// TwinCAT 3 PLC project JumpStart
// Title: Lift Template
// Company: FHNW
// Author: mbo
// ProjectVersion: 1.0.0
// ProgramVersion: 3.1.4026.20
// CompilerDefines: VISU_USEPROPERTYINFO
// libraries:
//   Tc2_Math, * (Beckhoff Automation GmbH)
//   Tc2_MC2, * (Beckhoff Automation GmbH)
//   Tc2_Standard, * (Beckhoff Automation GmbH)
//   Tc2_System, * (Beckhoff Automation GmbH)
//   Tc2_Utilities, * (Beckhoff Automation GmbH)
//   Tc3_IotBase, * (Beckhoff Automation GmbH)
//   Tc3_JsonXml, * (Beckhoff Automation GmbH)
//   VisuDialogs, * (System)
// project tree:
//   0_App/ IO_L1.TcGVL, IO_PLC.TcGVL, Divers.TcGVL, MAIN.TcPOU
//   0_App/Lib/Diverses/ ENUM_Achse.TcDUT, ENUM_Fahrsystem.TcDUT, ENUM_Tuer.TcDUT, FB_Logik_FIFO.TcPOU, FB_Logik_ShortestDistance.TcPOU, ITF_Fahrlogik.TcIO, ST_Error.TcDUT, ST_Fahrauftrag.TcDUT
//   0_App/Lib/ FB_Achse.TcPOU, FB_Blinker.TcPOU, FB_Fahrleitsystem.TcPOU, FB_Manuell.TcPOU, FB_Panel.TcPOU, FB_Taskmanager_1.TcPOU, FB_Tuer.TcPOU, FC_GetFloorPosition.TcPOU
//   7_Visu/Common/ Control.TcVIS, Floor.TcVIS, FloorControl.TcVIS, Lift.TcVIS, Lift_Axis.TcVIS, Lift_Floors.TcVIS, View_3Lifts.TcVIS
//   7_Visu/ Lift_1.TcVIS, Handbetrieb.TcVIS, Visu_Liftkabine.TcGVL, Visu_Liftkabine.TcVIS, Visu_Manuellmodus.TcGVL
//   9_Modell/Lib/ FB_MotionAxisPassive.TcPOU, FB_SimpleAxis.TcPOU, F_CycleTime.TcPOU, F_SpeedPerCycle.TcPOU
//   9_Modell/ MAIN_Modell.TcPOU, Visu_L1.TcGVL
//   / GlobalTextList.TcGTLO, PlcTask.TcTTO, Visualization Manager.TcVMO (not stored)
// real-time tasks:
//   TASK PlcTask: cycle T#10ms, priority 20, ADS port 350
// motion (NC):
//   TASK NC-Task 1 SAF: cycle T#2ms, priority 4, ADS port 501
//   TASK NC-Task 1 SVB: cycle T#10ms, priority 8, ADS port 511
//   AXIS Achse 1 - Lift1 (id 1)
//     Dynamic: Acceleration=1200, Deceleration=1200, Jerk=7200
//     Velo: FastManual=300, Maximum=500
//     OtherSettings: AllowMotionCmdToSlave=true
//     encoder EncType=4
//       EncPara: ScaleFactorNumerator=0.045066, MaxCount=#x0000ffff
//         Inc: RefSearchInverse=true, RefSyncInverse=false, RefMode=1, RefSoftSyncMask=#x0000ffff
//         TimeComp: TimeCompMode=1, EncDelayCycles=4
//     drive DrvType=23
//       DrvPara: Inverse=true
//         Analog: VeloReferenz=540, TorqueSetpointScale=10, ScaleFactorActTorque=0.1
//         TimeComp: TaskDelayCycles=1
//     controller CtrType=1
//       CtrPara: PriorControlFactor=1
//         PosDiffControl: Range=20
//         PID: PosKp=100
//         Observer: BandWidth=20
//   AXIS Achse 2 (id 2)
//     OtherSettings: AllowMotionCmdToSlave=true
//     encoder EncType=4
//       EncPara: MaxCount=#x0000ffff
//         Inc: RefSoftSyncMask=#x0000ffff
//     drive DrvType=23
//       Analog: TorqueSetpointScale=10, ScaleFactorActTorque=0.1
//       TimeComp: TaskDelayCycles=1
//     controller CtrType=1
//       CtrPara: PriorControlFactor=1
//         Observer: BandWidth=20
// I/O:
//   DEVICE Gerät 1 (EtherCAT), AmsNetId 192.168.10.51.2.1
//     Klemme 1 (EK1100) [EK1100 EtherCAT-Koppler (2A E-Bus)]
//       Klemme 2 (EL1262) [EL1262 2K. Dig. Eingang 24V, 1µs, DC Oversample]
//       Klemme 3 (EL2262) [EL2262 2K. Dig. Ausgang 24V, 1µs, DC Oversample]
//       Klemme 4 (EL1809) [EL1809 16K. Dig. Eingang 24V, 3ms]
//       Klemme 5 (EL2809) [EL2809 16K. Dig. Ausgang 24V, 0.5A]
//       Klemme 6 (EL3064) [EL3064 4K.Ana. Eingang 0-10V]
//       Klemme 7 (EL4004) [EL4004 4K. Ana. Ausgang 0-10V, 12bit]
//       Klemme 8 (EL5152) [EL5152 2K. Inc. Encoder]
//       Klemme 9 (EK1122) [EK1122 2-Port EtherCAT-Abzweig]
//       Klemme 10 (EL9011) [EL9011 Endklemme]
//   DEVICE Gerät 2 (EtherCAT), AmsNetId 192.168.10.51.3.1
//     Klemme 11 (EK1100) [EK1100 EtherCAT-Koppler (2A E-Bus)]
//       Klemme 12 (EL1809) [EL1809 16K. Dig. Eingang 24V, 3ms]
//       Klemme 13 (EL1809) [EL1809 16K. Dig. Eingang 24V, 3ms]
//       Klemme 14 (EL1809) [EL1809 16K. Dig. Eingang 24V, 3ms]
//       Klemme 15 (EL1809) [EL1809 16K. Dig. Eingang 24V, 3ms]
//       Klemme 16 (EL2809) [EL2809 16K. Dig. Ausgang 24V, 0.5A]
//       Klemme 17 (EL2809) [EL2809 16K. Dig. Ausgang 24V, 0.5A]
//       Klemme 18 (EL2809) [EL2809 16K. Dig. Ausgang 24V, 0.5A]
//       Klemme 19 (EL2809) [EL2809 16K. Dig. Ausgang 24V, 0.5A]
//       Klemme 20 (EL2809) [EL2809 16K. Dig. Ausgang 24V, 0.5A]
//       Klemme 21 (EL2809) [EL2809 16K. Dig. Ausgang 24V, 0.5A]
//       Klemme 22 (EL7342) [EL7342 2K. DC-Motor-Endstufe (50V, 3.5A)]
//       Klemme 37 (EL9011) [EL9011 Endklemme]
// variable links:
//   NC-Task 1 SAF/Axes/Achse 1 - Lift1 <-> Device 2 (EtherCAT)/Term 11 (EK1100)/Term 22 (EL7342)
//     Drive/Inputs/In/nState1 @bit 3 <-> DCM Status Channel 1/Status/Error
//     Drive/Inputs/In/nState1 @bit 5 <-> DCM Status Channel 1/Status/Moving negative
//     Drive/Inputs/In/nState1 @bit 4 <-> DCM Status Channel 1/Status/Moving positive
//     Drive/Inputs/In/nState1 @bit 1 <-> DCM Status Channel 1/Status/Ready
//     Drive/Inputs/In/nState1 <-> DCM Status Channel 1/Status/Ready to enable
//     Drive/Inputs/In/nState1 @bit 6 <-> DCM Status Channel 1/Status/Torque reduced
//     Drive/Inputs/In/nState1 @bit 2 <-> DCM Status Channel 1/Status/Warning
//     Drive/Inputs/In/nState2 @bit 4 <-> DCM Status Channel 1/Status/Digital input 2
//     Drive/Inputs/In/nState2 @bit 5 <-> DCM Status Channel 1/Status/Sync error
//     Drive/Inputs/In/nState2 @bit 7 <-> DCM Status Channel 1/Status/TxPDO Toggle
//     Drive/Inputs/In/nState4 @bit 1 <-> WcState/InputToggle
//     Drive/Inputs/In/nState4 <-> WcState/WcState
//     Drive/Outputs/Out/nCtrl1 <-> DCM Control Channel 1/Control/Enable
//     Drive/Outputs/Out/nCtrl1 @bit 2 <-> DCM Control Channel 1/Control/Reduce torque
//     Drive/Outputs/Out/nCtrl1 @bit 1 <-> DCM Control Channel 1/Control/Reset
//     Drive/Outputs/Out/nCtrl1 @bit 3 <-> DCM Control Channel 1/Control/Threshold active
//     Drive/Outputs/Out/nDataOut2[0] <-> DCM Velocity Channel 1/Velocity
//     Enc/Inputs/In/nDataIn1[0] <-> ENC Status compact Channel 1/Counter value
//     Enc/Inputs/In/nDataIn2[0] <-> ENC Status compact Channel 1/Latch value
//     Enc/Inputs/In/nState1 @bit 4 <-> ENC Status compact Channel 1/Status/Counter overflow
//     Enc/Inputs/In/nState1 @bit 3 <-> ENC Status compact Channel 1/Status/Counter underflow
//     Enc/Inputs/In/nState1 @bit 7 <-> ENC Status compact Channel 1/Status/Extrapolation stall
//     Enc/Inputs/In/nState1 @bit 1 <-> ENC Status compact Channel 1/Status/Latch extern valid
//     Enc/Inputs/In/nState1 @bit 2 <-> ENC Status compact Channel 1/Status/Set counter done
//     Enc/Inputs/In/nState2 @bit 4 <-> ENC Status compact Channel 1/Status/Status of extern latch
//     Enc/Inputs/In/nState2 <-> ENC Status compact Channel 1/Status/Status of input A
//     Enc/Inputs/In/nState2 @bit 1 <-> ENC Status compact Channel 1/Status/Status of input B
//     Enc/Inputs/In/nState2 @bit 5 <-> ENC Status compact Channel 1/Status/Sync error
//     Enc/Inputs/In/nState2 @bit 7 <-> ENC Status compact Channel 1/Status/TxPDO Toggle
//     Enc/Inputs/In/nState4 @bit 1 <-> WcState/InputToggle
//     Enc/Inputs/In/nState4 <-> WcState/WcState
//     Enc/Outputs/Out/nCtrl1 @bit 3 <-> ENC Control compact Channel 1/Control/Enable latch extern on negative edge
//     Enc/Outputs/Out/nCtrl1 @bit 1 <-> ENC Control compact Channel 1/Control/Enable latch extern on positive edge
//     Enc/Outputs/Out/nCtrl1 @bit 2 <-> ENC Control compact Channel 1/Control/Set counter
//     Enc/Outputs/Out/nDataOut1[0] <-> ENC Control compact Channel 1/Set counter value
//   NC-Task 1 SAF/Axes/Achse 2 <-> Device 2 (EtherCAT)/Term 11 (EK1100)/Term 22 (EL7342)
//     Drive/Inputs/In/nState1 @bit 3 <-> DCM Status Channel 2/Status/Error
//     Drive/Inputs/In/nState1 @bit 5 <-> DCM Status Channel 2/Status/Moving negative
//     Drive/Inputs/In/nState1 @bit 4 <-> DCM Status Channel 2/Status/Moving positive
//     Drive/Inputs/In/nState1 @bit 1 <-> DCM Status Channel 2/Status/Ready
//     Drive/Inputs/In/nState1 <-> DCM Status Channel 2/Status/Ready to enable
//     Drive/Inputs/In/nState1 @bit 6 <-> DCM Status Channel 2/Status/Torque reduced
//     Drive/Inputs/In/nState1 @bit 2 <-> DCM Status Channel 2/Status/Warning
//     Drive/Inputs/In/nState2 @bit 3 <-> DCM Status Channel 2/Status/Digital input 1
//     Drive/Inputs/In/nState2 @bit 4 <-> DCM Status Channel 2/Status/Digital input 2
//     Drive/Inputs/In/nState2 @bit 5 <-> DCM Status Channel 2/Status/Sync error
//     Drive/Inputs/In/nState2 @bit 7 <-> DCM Status Channel 2/Status/TxPDO Toggle
//     Drive/Inputs/In/nState4 @bit 1 <-> WcState/InputToggle
//     Drive/Inputs/In/nState4 <-> WcState/WcState
//     Drive/Outputs/Out/nCtrl1 <-> DCM Control Channel 2/Control/Enable
//     Drive/Outputs/Out/nCtrl1 @bit 2 <-> DCM Control Channel 2/Control/Reduce torque
//     Drive/Outputs/Out/nCtrl1 @bit 1 <-> DCM Control Channel 2/Control/Reset
//     Drive/Outputs/Out/nCtrl1 @bit 3 <-> DCM Control Channel 2/Control/Threshold active
//     Drive/Outputs/Out/nDataOut2[0] <-> DCM Velocity Channel 2/Velocity
//     Enc/Inputs/In/nDataIn1[0] <-> ENC Status compact Channel 2/Counter value
//     Enc/Inputs/In/nDataIn2[0] <-> ENC Status compact Channel 2/Latch value
//     Enc/Inputs/In/nState1 @bit 4 <-> ENC Status compact Channel 2/Status/Counter overflow
//     Enc/Inputs/In/nState1 @bit 3 <-> ENC Status compact Channel 2/Status/Counter underflow
//     Enc/Inputs/In/nState1 @bit 7 <-> ENC Status compact Channel 2/Status/Extrapolation stall
//     Enc/Inputs/In/nState1 @bit 1 <-> ENC Status compact Channel 2/Status/Latch extern valid
//     Enc/Inputs/In/nState1 @bit 2 <-> ENC Status compact Channel 2/Status/Set counter done
//     Enc/Inputs/In/nState2 @bit 4 <-> ENC Status compact Channel 2/Status/Status of extern latch
//     Enc/Inputs/In/nState2 <-> ENC Status compact Channel 2/Status/Status of input A
//     Enc/Inputs/In/nState2 @bit 1 <-> ENC Status compact Channel 2/Status/Status of input B
//     Enc/Inputs/In/nState2 @bit 5 <-> ENC Status compact Channel 2/Status/Sync error
//     Enc/Inputs/In/nState2 @bit 7 <-> ENC Status compact Channel 2/Status/TxPDO Toggle
//     Enc/Inputs/In/nState4 @bit 1 <-> WcState/InputToggle
//     Enc/Inputs/In/nState4 <-> WcState/WcState
//     Enc/Outputs/Out/nCtrl1 @bit 3 <-> ENC Control compact Channel 2/Control/Enable latch extern on negative edge
//     Enc/Outputs/Out/nCtrl1 @bit 1 <-> ENC Control compact Channel 2/Control/Enable latch extern on positive edge
//     Enc/Outputs/Out/nCtrl1 @bit 2 <-> ENC Control compact Channel 2/Control/Set counter
//     Enc/Outputs/Out/nDataOut1[0] <-> ENC Control compact Channel 2/Set counter value
//   JumpStart Instance <-> Device 1 (EtherCAT)/Term 1 (EK1100)/Term 4 (EL1809)
//     PlcTask Inputs/IO_PLC.T1 <-> Channel 15/Input
//     PlcTask Inputs/IO_PLC.T2 <-> Channel 16/Input
//   JumpStart Instance <-> Device 1 (EtherCAT)/Term 1 (EK1100)/Term 5 (EL2809)
//     PlcTask Outputs/IO_PLC.LED_Green <-> Channel 14/Output
//     PlcTask Outputs/IO_PLC.LED_Red <-> Channel 16/Output
//     PlcTask Outputs/IO_PLC.LED_Yellow <-> Channel 15/Output
//   JumpStart Instance <-> Device 1 (EtherCAT)/Term 1 (EK1100)/Term 6 (EL3064)
//     PlcTask Inputs/IO_PLC.P <-> AI Standard Channel 4/Value
//   JumpStart Instance <-> Device 2 (EtherCAT)/Term 11 (EK1100)/Term 12 (EL1809)
//     PlcTask Inputs/IO_L1.Panel_1_Btn[1] <-> Channel 1/Input
//     PlcTask Inputs/IO_L1.Panel_1_Btn[2] <-> Channel 2/Input
//     PlcTask Inputs/IO_L1.Panel_1_Btn[3] <-> Channel 3/Input
//     PlcTask Inputs/IO_L1.Panel_1_Btn[4] <-> Channel 4/Input
//     PlcTask Inputs/IO_L1.Panel_1_Btn[5] <-> Channel 5/Input
//     PlcTask Inputs/IO_L1.Panel_1_Btn[6] <-> Channel 6/Input
//     PlcTask Inputs/IO_L1.Panel_2_Btn[1] <-> Channel 7/Input
//     PlcTask Inputs/IO_L1.Panel_2_Btn[2] <-> Channel 8/Input
//     PlcTask Inputs/IO_L1.Panel_2_Btn[3] <-> Channel 9/Input
//     PlcTask Inputs/IO_L1.Panel_2_Btn[4] <-> Channel 10/Input
//     PlcTask Inputs/IO_L1.Panel_2_Btn[5] <-> Channel 11/Input
//     PlcTask Inputs/IO_L1.Panel_2_Btn[6] <-> Channel 12/Input
//     PlcTask Inputs/IO_L1.Panel_3_Btn[1] <-> Channel 13/Input
//     PlcTask Inputs/IO_L1.Panel_3_Btn[2] <-> Channel 14/Input
//     PlcTask Inputs/IO_L1.Panel_3_Btn[3] <-> Channel 15/Input
//     PlcTask Inputs/IO_L1.Panel_3_Btn[4] <-> Channel 16/Input
//   JumpStart Instance <-> Device 2 (EtherCAT)/Term 11 (EK1100)/Term 13 (EL1809)
//     PlcTask Inputs/IO_L1.Panel_3_Btn[5] <-> Channel 1/Input
//     PlcTask Inputs/IO_L1.Panel_3_Btn[6] <-> Channel 2/Input
//     PlcTask Inputs/IO_L1.Panel_4_Btn[1] <-> Channel 3/Input
//     PlcTask Inputs/IO_L1.Panel_4_Btn[2] <-> Channel 4/Input
//     PlcTask Inputs/IO_L1.Panel_4_Btn[3] <-> Channel 5/Input
//     PlcTask Inputs/IO_L1.Panel_4_Btn[4] <-> Channel 6/Input
//     PlcTask Inputs/IO_L1.Panel_4_Btn[5] <-> Channel 7/Input
//     PlcTask Inputs/IO_L1.Panel_4_Btn[6] <-> Channel 8/Input
//     PlcTask Inputs/IO_L1.Panel_5_Btn[1] <-> Channel 9/Input
//     PlcTask Inputs/IO_L1.Panel_5_Btn[2] <-> Channel 10/Input
//     PlcTask Inputs/IO_L1.Panel_5_Btn[3] <-> Channel 11/Input
//     PlcTask Inputs/IO_L1.Panel_5_Btn[4] <-> Channel 12/Input
//     PlcTask Inputs/IO_L1.Panel_5_Btn[5] <-> Channel 13/Input
//     PlcTask Inputs/IO_L1.Panel_5_Btn[6] <-> Channel 14/Input
//     PlcTask Inputs/IO_L1.Panel_6_Btn[1] <-> Channel 15/Input
//     PlcTask Inputs/IO_L1.Panel_6_Btn[2] <-> Channel 16/Input
//   JumpStart Instance <-> Device 2 (EtherCAT)/Term 11 (EK1100)/Term 14 (EL1809)
//     PlcTask Inputs/IO_L1.Door_{1..6}_SensorClosed <-> Channel {5..15 step 2}/Input  (6 links)
//     PlcTask Inputs/IO_L1.Door_{1..6}_SensorOpen <-> Channel {6..16 step 2}/Input  (6 links)
//     PlcTask Inputs/IO_L1.Panel_6_Btn[{3..6}] <-> Channel {1..4}/Input  (4 links)
//   JumpStart Instance <-> Device 2 (EtherCAT)/Term 11 (EK1100)/Term 15 (EL1809)
//     PlcTask Inputs/IO_L1.Control_Automatic <-> Channel 2/Input
//     PlcTask Inputs/IO_L1.Control_EmergencyStopActive <-> Channel 12/Input
//     PlcTask Inputs/IO_L1.Control_Manual <-> Channel 1/Input
//     PlcTask Inputs/IO_L1.Control_Overload <-> Channel 5/Input
//     PlcTask Inputs/IO_L1.Control_Reset <-> Channel 3/Input
//     PlcTask Inputs/IO_L1.Control_Start <-> Channel 4/Input
//     PlcTask Inputs/IO_L1.Door_{1..6}_SensorActive <-> Channel {6..11}/Input  (6 links)
//   JumpStart Instance <-> Device 2 (EtherCAT)/Term 11 (EK1100)/Term 16 (EL2809)
//     PlcTask Outputs/IO_L1.Panel_1_BCD_Bit[{0..3}] <-> Channel {7..10}/Output  (4 links)
//     PlcTask Outputs/IO_L1.Panel_1_BtnLed[1] <-> Channel 1/Output
//     PlcTask Outputs/IO_L1.Panel_1_BtnLed[2] <-> Channel 2/Output
//     PlcTask Outputs/IO_L1.Panel_1_BtnLed[3] <-> Channel 3/Output
//     PlcTask Outputs/IO_L1.Panel_1_BtnLed[4] <-> Channel 4/Output
//     PlcTask Outputs/IO_L1.Panel_1_BtnLed[5] <-> Channel 5/Output
//     PlcTask Outputs/IO_L1.Panel_1_BtnLed[6] <-> Channel 6/Output
//     PlcTask Outputs/IO_L1.Panel_2_BtnLed[1] <-> Channel 13/Output
//     PlcTask Outputs/IO_L1.Panel_2_BtnLed[2] <-> Channel 14/Output
//     PlcTask Outputs/IO_L1.Panel_2_BtnLed[3] <-> Channel 15/Output
//     PlcTask Outputs/IO_L1.Panel_2_BtnLed[4] <-> Channel 16/Output
//     PlcTask Outputs/IO_L1.Panel_1_Led_Down <-> Channel 12/Output
//     PlcTask Outputs/IO_L1.Panel_1_Led_Up <-> Channel 11/Output
//   JumpStart Instance <-> Device 2 (EtherCAT)/Term 11 (EK1100)/Term 17 (EL2809)
//     PlcTask Outputs/IO_L1.Panel_2_BCD_Bit[0] <-> Channel 3/Output
//     PlcTask Outputs/IO_L1.Panel_2_BCD_Bit[1] <-> Channel 4/Output
//     PlcTask Outputs/IO_L1.Panel_2_BCD_Bit[2] <-> Channel 5/Output
//     PlcTask Outputs/IO_L1.Panel_2_BCD_Bit[3] <-> Channel 6/Output
//     PlcTask Outputs/IO_L1.Panel_3_BCD_Bit[0] <-> Channel 15/Output
//     PlcTask Outputs/IO_L1.Panel_3_BCD_Bit[1] <-> Channel 16/Output
//     PlcTask Outputs/IO_L1.Panel_2_BtnLed[5] <-> Channel 1/Output
//     PlcTask Outputs/IO_L1.Panel_2_BtnLed[6] <-> Channel 2/Output
//     PlcTask Outputs/IO_L1.Panel_3_BtnLed[1] <-> Channel 9/Output
//     PlcTask Outputs/IO_L1.Panel_3_BtnLed[2] <-> Channel 10/Output
//     PlcTask Outputs/IO_L1.Panel_3_BtnLed[3] <-> Channel 11/Output
//     PlcTask Outputs/IO_L1.Panel_3_BtnLed[4] <-> Channel 12/Output
//     PlcTask Outputs/IO_L1.Panel_3_BtnLed[5] <-> Channel 13/Output
//     PlcTask Outputs/IO_L1.Panel_3_BtnLed[6] <-> Channel 14/Output
//     PlcTask Outputs/IO_L1.Panel_2_Led_Down <-> Channel 8/Output
//     PlcTask Outputs/IO_L1.Panel_2_Led_Up <-> Channel 7/Output
//   JumpStart Instance <-> Device 2 (EtherCAT)/Term 11 (EK1100)/Term 18 (EL2809)
//     PlcTask Outputs/IO_L1.Panel_3_BCD_Bit[2] <-> Channel 1/Output
//     PlcTask Outputs/IO_L1.Panel_3_BCD_Bit[3] <-> Channel 2/Output
//     PlcTask Outputs/IO_L1.Panel_4_BCD_Bit[0] <-> Channel 11/Output
//     PlcTask Outputs/IO_L1.Panel_4_BCD_Bit[1] <-> Channel 12/Output
//     PlcTask Outputs/IO_L1.Panel_4_BCD_Bit[2] <-> Channel 13/Output
//     PlcTask Outputs/IO_L1.Panel_4_BCD_Bit[3] <-> Channel 14/Output
//     PlcTask Outputs/IO_L1.Panel_3_Led_Down <-> Channel 4/Output
//     PlcTask Outputs/IO_L1.Panel_4_Led_Down <-> Channel 16/Output
//     PlcTask Outputs/IO_L1.Panel_3_Led_Up <-> Channel 3/Output
//     PlcTask Outputs/IO_L1.Panel_4_Led_Up <-> Channel 15/Output
//     PlcTask Outputs/IO_L1.Panel_4_BtnLed[{1..6}] <-> Channel {5..10}/Output  (6 links)
//   JumpStart Instance <-> Device 2 (EtherCAT)/Term 11 (EK1100)/Term 19 (EL2809)
//     PlcTask Outputs/IO_L1.Panel_5_BCD_Bit[{0..3}] <-> Channel {7..10}/Output  (4 links)
//     PlcTask Outputs/IO_L1.Panel_5_BtnLed[1] <-> Channel 1/Output
//     PlcTask Outputs/IO_L1.Panel_5_BtnLed[2] <-> Channel 2/Output
//     PlcTask Outputs/IO_L1.Panel_5_BtnLed[3] <-> Channel 3/Output
//     PlcTask Outputs/IO_L1.Panel_5_BtnLed[4] <-> Channel 4/Output
//     PlcTask Outputs/IO_L1.Panel_5_BtnLed[5] <-> Channel 5/Output
//     PlcTask Outputs/IO_L1.Panel_5_BtnLed[6] <-> Channel 6/Output
//     PlcTask Outputs/IO_L1.Panel_6_BtnLed[1] <-> Channel 13/Output
//     PlcTask Outputs/IO_L1.Panel_6_BtnLed[2] <-> Channel 14/Output
//     PlcTask Outputs/IO_L1.Panel_6_BtnLed[3] <-> Channel 15/Output
//     PlcTask Outputs/IO_L1.Panel_6_BtnLed[4] <-> Channel 16/Output
//     PlcTask Outputs/IO_L1.Panel_5_Led_Down <-> Channel 12/Output
//     PlcTask Outputs/IO_L1.Panel_5_Led_Up <-> Channel 11/Output
//   JumpStart Instance <-> Device 2 (EtherCAT)/Term 11 (EK1100)/Term 20 (EL2809)
//     PlcTask Outputs/IO_L1.Door_{1..4}_MotorClose <-> Channel {10..16 step 2}/Output  (4 links)
//     PlcTask Outputs/IO_L1.Door_{1..4}_MotorOpen <-> Channel {9..15 step 2}/Output  (4 links)
//     PlcTask Outputs/IO_L1.Panel_6_BCD_Bit[{0..3}] <-> Channel {3..6}/Output  (4 links)
//     PlcTask Outputs/IO_L1.Panel_6_BtnLed[5] <-> Channel 1/Output
//     PlcTask Outputs/IO_L1.Panel_6_BtnLed[6] <-> Channel 2/Output
//     PlcTask Outputs/IO_L1.Panel_6_Led_Down <-> Channel 8/Output
//     PlcTask Outputs/IO_L1.Panel_6_Led_Up <-> Channel 7/Output
//   JumpStart Instance <-> Device 2 (EtherCAT)/Term 11 (EK1100)/Term 21 (EL2809)
//     PlcTask Outputs/IO_L1.Control_LED_Blue <-> Channel 7/Output
//     PlcTask Outputs/IO_L1.Control_LED_Red <-> Channel 6/Output
//     PlcTask Outputs/IO_L1.Control_LED_White <-> Channel 8/Output
//     PlcTask Outputs/IO_L1.Control_LED_Yellow <-> Channel 5/Output
//     PlcTask Outputs/IO_L1.Door_5_MotorClose <-> Channel 2/Output
//     PlcTask Outputs/IO_L1.Door_6_MotorClose <-> Channel 4/Output
//     PlcTask Outputs/IO_L1.Door_5_MotorOpen <-> Channel 1/Output
//     PlcTask Outputs/IO_L1.Door_6_MotorOpen <-> Channel 3/Output
//   JumpStart Instance <-> Device 2 (EtherCAT)/Term 11 (EK1100)/Term 22 (EL7342)
//     PlcTask Inputs/IO_L1.Control_LiftAxisReference <-> DCM Status Channel 1/Status/Digital input 1
//   JumpStart Instance <-> NC-Task 1 SAF/Axes/Achse 1 - Lift1
//     PlcTask Inputs/IO_L1.LiftAxis.NcToPlc <-> Outputs/ToPlc
//     PlcTask Outputs/IO_L1.LiftAxis.PlcToNc <-> Inputs/FromPlc

CONFIGURATION JumpStart
    RESOURCE PLC ON TwinCAT3
        TASK PlcTask(INTERVAL := T#10ms, PRIORITY := 20);
        PROGRAM MAIN_Modell WITH PlcTask : MAIN_Modell;
        PROGRAM MAIN WITH PlcTask : MAIN;
    END_RESOURCE
END_CONFIGURATION

// ---- 0_App/Lib/Diverses/ENUM_Achse.TcDUT
{attribute 'qualified_only'}
{attribute 'strict'}
{attribute 'to_string'}
TYPE ENUM_Achse :
(
	PowerOn := 1,
	Referenzieren := 2,
	Warten := 0,
	Positionieren := 3,
	Error := 4
	
	
);
END_TYPE

// ---- 0_App/Lib/Diverses/ENUM_Fahrsystem.TcDUT
{attribute 'qualified_only'}
{attribute 'strict'}
{attribute 'to_string'}
TYPE ENUM_Fahrsystem :
(
	Warten := 0,
	Sicherheitscheck := 1,
	ZumStartStockwerk := 2,
	Tueren := 3,
	ZumZielStockwerk := 4,
	Aufstartablauf := 5
);
END_TYPE

// ---- 0_App/Lib/Diverses/ENUM_Tuer.TcDUT
{attribute 'qualified_only'}
{attribute 'strict'}
{attribute 'to_string'}
TYPE ENUM_Tuer :
(
	
    TuereZu,
    TuereOeffnen,
    TuereAuf,
    TuereSchliessen,
    Error
);
END_TYPE

// ---- 0_App/Lib/Diverses/ST_Error.TcDUT
TYPE ST_Error :
STRUCT
    // Achse
    AchsePower      : BOOL;
    AchseHome       : BOOL;
    AchseMove       : BOOL;
    AchseJog        : BOOL;
    AchseFehlercode : UDINT;

    // Türen
    TuerTimeout     : ARRAY[1..6] OF BOOL;

    // Allgemein
    NotAus          : BOOL;
    Brandalarm      : BOOL;

    // Zusammengefasst — wird automatisch berechnet
    IrgendeinFehler : BOOL;
    IrgendEineWarnung : BOOL;
    FehlerQuittiert : BOOL;
END_STRUCT
END_TYPE

// ---- 0_App/Lib/Diverses/ST_Fahrauftrag.TcDUT
TYPE ST_Fahrauftrag :
STRUCT
	Startstockwerk : INT;
	Zielstockwerk : INT;
	istAktiv : BOOL;
	Auftragsnummer : DINT;
END_STRUCT
END_TYPE

// ---- 0_App/IO_L1.TcGVL
{attribute 'qualified_only'}
VAR_GLOBAL
	LiftAxis					: AXIS_REF;
	
	Door_1_SensorOpen			AT %I*	: BOOL;	// Door level 1 open
	Door_1_SensorClosed  		AT %I*	: BOOL; // Door level 1 closed
	Door_1_SensorActive			AT %I*	: BOOL; // Door level 1 sensor active
	Door_1_MotorOpen			AT %Q* 	: BOOL; // Motor level 1 - Open
	Door_1_MotorClose			AT %Q* 	: BOOL; // Motor level 1 - Close
	
	Panel_1_Btn					AT %I*  : ARRAY[1..6] OF BOOL; // Panel Level 1 - Buttons
	Panel_1_BtnLed				AT %Q*  : ARRAY[1..6] OF BOOL; // Panel Level 1 - Button LEDs
	Panel_1_Led_Up				AT %Q*  : BOOL; // Panel Level 1 - Led Up
	Panel_1_Led_Down			AT %Q*  : BOOL; // Panel Level 1 - Led Down
	Panel_1_BCD_Bit				AT %Q* 	: ARRAY[0..3] OF BOOL; // Panel Level 1- BCD Bit 0..3
	
	Door_2_SensorOpen			AT %I*	: BOOL;	// Door level 2 open
	Door_2_SensorClosed  		AT %I*	: BOOL; // Door level 2 closed
	Door_2_SensorActive			AT %I*	: BOOL; // Door level 2 sensor active
	Door_2_MotorOpen			AT %Q* 	: BOOL; // Motor level 2 - Open
	Door_2_MotorClose			AT %Q* 	: BOOL; // Motor level 2 - Close
	
	Panel_2_Btn					AT %I*  : ARRAY[1..6] OF BOOL; // Panel Level 2 - Buttons
	Panel_2_BtnLed				AT %Q*  : ARRAY[1..6] OF BOOL; // Panel Level 2 - Button LEDs
	Panel_2_Led_Up				AT %Q*  : BOOL; // Panel Level 2 - Led Up
	Panel_2_Led_Down			AT %Q*  : BOOL; // Panel Level 2 - Led Down
	Panel_2_BCD_Bit				AT %Q* 	: ARRAY[0..3] OF BOOL; // Panel Level 2- BCD Bit 0..3
	
	Door_3_SensorOpen			AT %I*	: BOOL;	// Door level 3 open
	Door_3_SensorClosed  		AT %I*	: BOOL; // Door level 3 closed
	Door_3_SensorActive			AT %I*	: BOOL; // Door level 3 sensor active
	Door_3_MotorOpen			AT %Q* 	: BOOL; // Motor level 3 - Open
	Door_3_MotorClose			AT %Q* 	: BOOL; // Motor level 3 - Close
	
	Panel_3_Btn					AT %I*  : ARRAY[1..6] OF BOOL; // Panel Level 3 - Buttons
	Panel_3_BtnLed				AT %Q*  : ARRAY[1..6] OF BOOL; // Panel Level 3 - Button LEDs
	Panel_3_Led_Up				AT %Q*  : BOOL; // Panel Level 3 - Led Up
	Panel_3_Led_Down			AT %Q*  : BOOL; // Panel Level 3 - Led Down
	Panel_3_BCD_Bit				AT %Q* 	: ARRAY[0..3] OF BOOL; // Panel Level 3- BCD Bit 0..3
	
	
	Door_4_SensorOpen			AT %I*	: BOOL;	// Door level 4 open
	Door_4_SensorClosed  		AT %I*	: BOOL; // Door level 4 closed
	Door_4_SensorActive			AT %I*	: BOOL; // Door level 4 sensor active
	Door_4_MotorOpen			AT %Q* 	: BOOL; // Motor level 4 - Open
	Door_4_MotorClose			AT %Q* 	: BOOL; // Motor level 4 - Close
	
	Panel_4_Btn					AT %I*  : ARRAY[1..6] OF BOOL; // Panel Level 4 - Buttons
	Panel_4_BtnLed				AT %Q*  : ARRAY[1..6] OF BOOL; // Panel Level 4 - Button LEDs
	Panel_4_Led_Up				AT %Q*  : BOOL; // Panel Level 4 - Led Up
	Panel_4_Led_Down			AT %Q*  : BOOL; // Panel Level 4 - Led Down
	Panel_4_BCD_Bit				AT %Q* 	: ARRAY[0..3] OF BOOL; // Panel Level 4- BCD Bit 0..3
	
	
	Door_5_SensorOpen			AT %I*	: BOOL;	// Door level 5 open
	Door_5_SensorClosed  		AT %I*	: BOOL; // Door level 5 closed
	Door_5_SensorActive			AT %I*	: BOOL; // Door level 5 sensor active
	Door_5_MotorOpen			AT %Q* 	: BOOL; // Motor level 5 - Open
	Door_5_MotorClose			AT %Q* 	: BOOL; // Motor level 5 - Close
	
	Panel_5_Btn					AT %I*  : ARRAY[1..6] OF BOOL; // Panel Level 5 - Buttons
	Panel_5_BtnLed				AT %Q*  : ARRAY[1..6] OF BOOL; // Panel Level 5 - Button LEDs
	Panel_5_Led_Up				AT %Q*  : BOOL; // Panel Level 5 - Led Up
	Panel_5_Led_Down			AT %Q*  : BOOL; // Panel Level 5 - Led Down
	Panel_5_BCD_Bit				AT %Q* 	: ARRAY[0..3] OF BOOL; // Panel Level 5- BCD Bit 0..3
	
	
	Door_6_SensorOpen			AT %I*	: BOOL;	// Door level 6 open
	Door_6_SensorClosed  		AT %I*	: BOOL; // Door level 6 closed
	Door_6_SensorActive			AT %I*	: BOOL; // Door level 6 sensor active
	Door_6_MotorOpen			AT %Q* 	: BOOL; // Motor level 6 - Open
	Door_6_MotorClose			AT %Q* 	: BOOL; // Motor level 6 - Close

	Panel_6_Btn					AT %I*  : ARRAY[1..6] OF BOOL; // Panel Level 6 - Buttons
	Panel_6_BtnLed				AT %Q*  : ARRAY[1..6] OF BOOL; // Panel Level 6 - Button LEDs
	Panel_6_Led_Up				AT %Q*  : BOOL; // Panel Level 6 - Led Up
	Panel_6_Led_Down			AT %Q*  : BOOL; // Panel Level 6 - Led Down
	Panel_6_BCD_Bit				AT %Q* 	: ARRAY[0..3] OF BOOL; // Panel Level 6- BCD Bit 0..3
	
	

	Control_Manual					AT %I*	: BOOL; // Mode: Manual
	Control_Automatic				AT %I*	: BOOL; // Mode: Automatic
	Control_Reset					AT %I*	: BOOL; // Reset
	Control_Start					AT %I*	: BOOL; // Start
	Control_EmergencyStopActive 	AT %I*	: BOOL; // Emergency stop active
	Control_Overload				AT %I*	: BOOL; // Lift overload
	Control_LiftAxisReference		AT %I*  : BOOL; // Lift reference sensor bottom
	Control_Firealarm				AT %I*  : BOOL; // Fire alarm signal
	
	Control_LED_Yellow				AT %Q*	: BOOL; // LED Yellow 
	Control_LED_Red					AT %Q*	: BOOL; // LED Red 
	Control_LED_Blue				AT %Q*	: BOOL; // LED Blue 
	Control_LED_White				AT %Q*	: BOOL; // LED White 
END_VAR

// ---- 0_App/IO_PLC.TcGVL
{attribute 'qualified_only'}
VAR_GLOBAL
	T1				AT %I*	: BOOL; 
	T2				AT %I*	: BOOL; 
	P				AT %I*	: INT; 	
	LED_Green 		AT %Q* : BOOL;
	LED_Yellow 		AT %Q* : BOOL;
	LED_Red 		AT %Q* : BOOL;
END_VAR

// ---- 0_App/Divers.TcGVL

VAR_GLOBAL
	NextfreeOrderID : INT;
	AktuellesStockwerk : INT;
	AktuellePosmm : LREAL;
	AutomatikmodusAktiv : BOOL;
	ManuellmodusAktiv : BOOL;
	AlleTuerenZu : BOOL;
	AchseSicher : BOOL;
	Fehler : ST_Error;
	Fehlertext : STRING(500);
END_VAR

// ---- 7_Visu/Visu_Liftkabine.TcGVL
{attribute 'qualified_only'}
VAR_GLOBAL
	TuerAuf : BOOL;
	TuerZu : BOOL;
	AktuellerStock : INT;
	
END_VAR

// ---- 7_Visu/Visu_Manuellmodus.TcGVL
{attribute 'qualified_only'}
VAR_GLOBAL
	AktuellePosmm : LREAL;
	JogAuf : BOOL;
	JogAb : BOOL;
	Zielstock : INT;
	PosAnfahren : BOOL;
	ReferenzStart : BOOL;
	bTuerAuf : ARRAY[1..6] OF BOOL;
	bTuerZu : ARRAY[1..6] OF BOOL;
	AlleTuerenZu : BOOL;
	AlleTuerenAuf : BOOL;
	adwFloorBtnColor : ARRAY[1..6] OF DWORD;

	adwTuerAufColor : ARRAY[1..6] OF DWORD;
	adwTuerZuColor  : ARRAY[1..6] OF DWORD;
	
END_VAR

// ---- 9_Modell/Visu_L1.TcGVL
{attribute 'qualified_only'}
VAR_GLOBAL
	Position_LIFT	: LREAL; // 0-100
	Door_1_Position	: REAL;
	Door_1_M_Open	: BOOL;
	Door_1_M_Close	: BOOL;
	Door_2_Position	: REAL;
	
	Door_2_M_Open	: BOOL;
	Door_2_M_Close	: BOOL;
	Door_3_Position	: REAL;
	
	Door_3_M_Open	: BOOL;
	Door_3_M_Close	: BOOL;
	Door_4_Position	: REAL;
	
	Door_4_M_Open	: BOOL;
	Door_4_M_Close	: BOOL;
	Door_5_Position	: REAL;
	
	Door_5_M_Open	: BOOL;
	Door_5_M_Close	: BOOL;
	Door_6_Position	: REAL;
	
	Door_6_M_Open	: BOOL;
	Door_6_M_Close	: BOOL;
	Color : DWORD := 16#FFFFA500;	

	Door_1_SensorOpen				: BOOL;	// Door level 1 open
	Door_1_SensorClosed  			: BOOL; // Door level 1 closed
	Door_1_SensorActive				: BOOL := TRUE; // Door level 1 sensor active
	Door_1_MotorOpen			 	: BOOL; // Motor level 1 - Open
	Door_1_MotorClose			 	: BOOL; // Motor level 1 - Close
	
	Panel_1_Btn					  : ARRAY[1..6] OF BOOL; // Panel Level 1 - Buttons
	Panel_1_BtnLed				  : ARRAY[1..6] OF BOOL; // Panel Level 1 - Button LEDs
	Panel_1_Led_Up				  : BOOL; // Panel Level 1 - Led Up
	Panel_1_Led_Down			  : BOOL; // Panel Level 1 - Led Down
	Panel_1_FloorNumber			 	: INT; // Panel Level 1 - Floor Number
	
	Door_2_SensorOpen				: BOOL;	// Door level 2 open
	Door_2_SensorClosed  			: BOOL; // Door level 2 closed
	Door_2_SensorActive				: BOOL := TRUE; // Door level 2 sensor active
	Door_2_MotorOpen			 	: BOOL; // Motor level 2 - Open
	Door_2_MotorClose			 	: BOOL; // Motor level 2 - Close
	
	Panel_2_Btn					  : ARRAY[1..6] OF BOOL; // Panel Level 2 - Buttons
	Panel_2_BtnLed				  : ARRAY[1..6] OF BOOL; // Panel Level 2 - Button LEDs
	Panel_2_Led_Up				  : BOOL; // Panel Level 2 - Led Up
	Panel_2_Led_Down			  : BOOL; // Panel Level 2 - Led Down
	Panel_2_FloorNumber			 	: INT; // Panel Level 2 - Floor Number
	
	Door_3_SensorOpen				: BOOL;	// Door level 3 open
	Door_3_SensorClosed  			: BOOL; // Door level 3 closed
	Door_3_SensorActive				: BOOL := TRUE; // Door level 3 sensor active
	Door_3_MotorOpen			 	: BOOL; // Motor level 3 - Open
	Door_3_MotorClose			 	: BOOL; // Motor level 3 - Close
	
	Panel_3_Btn					  : ARRAY[1..6] OF BOOL; // Panel Level 3 - Buttons
	Panel_3_BtnLed				  : ARRAY[1..6] OF BOOL; // Panel Level 3 - Button LEDs
	Panel_3_Led_Up				  : BOOL; // Panel Level 3 - Led Up
	Panel_3_Led_Down			  : BOOL; // Panel Level 3 - Led Down
	Panel_3_FloorNumber			 	: INT; // Panel Level 3 - Floor Number
	
	Door_4_SensorOpen				: BOOL;	// Door level 4 open
	Door_4_SensorClosed  			: BOOL; // Door level 4 closed
	Door_4_SensorActive				: BOOL := TRUE; // Door level 4 sensor active
	Door_4_MotorOpen			 	: BOOL; // Motor level 4 - Open
	Door_4_MotorClose			 	: BOOL; // Motor level 4 - Close
	
	Panel_4_Btn					  : ARRAY[1..6] OF BOOL; // Panel Level 4 - Buttons
	Panel_4_BtnLed				  : ARRAY[1..6] OF BOOL; // Panel Level 4 - Button LEDs
	Panel_4_Led_Up				  : BOOL; // Panel Level 4 - Led Up
	Panel_4_Led_Down			  : BOOL; // Panel Level 4 - Led Down
	Panel_4_FloorNumber			 	: INT; // Panel Level 4 - Floor Number
	
	Door_5_SensorOpen				: BOOL;	// Door level 5 open
	Door_5_SensorClosed  			: BOOL; // Door level 5 closed
	Door_5_SensorActive				: BOOL := TRUE; // Door level 5 sensor active
	Door_5_MotorOpen			 	: BOOL; // Motor level 5 - Open
	Door_5_MotorClose			 	: BOOL; // Motor level 5 - Close
	
	Panel_5_Btn					  : ARRAY[1..6] OF BOOL; // Panel Level 5 - Buttons
	Panel_5_BtnLed				  : ARRAY[1..6] OF BOOL; // Panel Level 5 - Button LEDs
	Panel_5_Led_Up				  : BOOL; // Panel Level 5 - Led Up
	Panel_5_Led_Down			  : BOOL; // Panel Level 5 - Led Down
	Panel_5_FloorNumber			 	: INT; // Panel Level 5 - Floor Number
	
	Door_6_SensorOpen				: BOOL;	// Door level 6 open
	Door_6_SensorClosed  			: BOOL; // Door level 6 closed
	Door_6_SensorActive				: BOOL := TRUE; // Door level 6 sensor active
	Door_6_MotorOpen			 	: BOOL; // Motor level 6 - Open
	Door_6_MotorClose			 	: BOOL; // Motor level 6 - Close

	Panel_6_Btn					  : ARRAY[1..6] OF BOOL; // Panel Level 6 - Buttons
	Panel_6_BtnLed				  : ARRAY[1..6] OF BOOL; // Panel Level 6 - Button LEDs
	Panel_6_Led_Up				  : BOOL; // Panel Level 6 - Led Up
	Panel_6_Led_Down			  : BOOL; // Panel Level 6 - Led Down
	Panel_6_FloorNumber			 	: INT; // Panel Level 6 - Floor Number
	
	Control_State						: INT;
	Control_Reset						: BOOL; // Reset
	Control_Start						: BOOL; // Start
	Control_EmergencyStopActive 		: BOOL; // Emergency stop active
	Control_Overload					: BOOL; // Lift overload
	Control_LiftAxisReference		  : BOOL; // Lift reference sensor bottom
	Control_Firealarm				  : BOOL; // Fire alarm signal
	
	Control_LED_Yellow					: BOOL; // LED Yellow 
	Control_LED_Red						: BOOL; // LED Red 
	Control_LED_Blue					: BOOL; // LED Blue 
	Control_LED_White					: BOOL; // LED White 
END_VAR

// ---- 0_App/Lib/Diverses/ITF_Fahrlogik.TcIO
INTERFACE ITF_Fahrlogik

METHOD M_getNextTask : ST_Fahrauftrag
VAR_INPUT
	LiftStockwerkAktuell : INT;
END_VAR
VAR_IN_OUT
    Auftraege : ARRAY[1..10] OF ST_Fahrauftrag; // Die Liste zum Durchsuchen
END_VAR
END_METHOD

END_INTERFACE

// ---- 9_Modell/MAIN_Modell.TcPOU
PROGRAM MAIN_Modell
VAR
	fbL1_Axis : FB_MotionAxisPassive;
	fbL1_Door_1	: FB_SimpleAxis;
	fbL1_Door_2	: FB_SimpleAxis;
	fbL1_Door_3	: FB_SimpleAxis;
	fbL1_Door_4	: FB_SimpleAxis;
	fbL1_Door_5	: FB_SimpleAxis;
	fbL1_Door_6	: FB_SimpleAxis;
	
END_VAR
VAR CONSTANT
	LIFT_CAP_HEIGHT : INT := 140;
	LIFT_DRIVE_AXIS : INT := 1460;
	LIFT_REF_SENSOR_POSITION : INT := 45;
END_VAR



fbL1_Axis(
	Axis := IO_L1.LiftAxis, 
	Length := LIFT_DRIVE_AXIS - LIFT_CAP_HEIGHT, 
	RefSensorPositionAbs := LIFT_REF_SENSOR_POSITION, 
	CurrentPosition => , 
	RefSensor => );
	
IO_L1.Control_LiftAxisReference := fbL1_Axis.RefSensor;
Visu_L1.Control_LiftAxisReference := fbL1_Axis.RefSensor;

fbL1_Door_1(
	MotorOpen:= IO_L1.Door_1_MotorOpen, 
	MotorClose:= IO_L1.Door_1_MotorClose,
	Position=> );
	
IO_L1.Door_1_SensorOpen := fbL1_Door_1.SensorOpenActive;
IO_L1.Door_1_SensorClosed := fbL1_Door_1.SensorCloseActive;
IO_L1.Door_1_SensorActive := Visu_L1.Door_1_SensorActive;

Visu_l1.Door_1_SensorOpen := IO_L1.Door_1_SensorOpen;
Visu_l1.Door_1_SensorClosed := IO_L1.Door_1_SensorClosed;
Visu_l1.Door_1_M_Open := IO_L1.Door_1_MotorOpen;
Visu_l1.Door_1_M_Close := IO_L1.Door_1_MotorClose;

fbL1_Door_2(
	MotorOpen:= IO_L1.Door_2_MotorOpen, 
	MotorClose:= IO_L1.Door_2_MotorClose,
	Position=> );
	
IO_L1.Door_2_SensorOpen := fbL1_Door_2.SensorOpenActive;
IO_L1.Door_2_SensorClosed := fbL1_Door_2.SensorCloseActive;
IO_L1.Door_2_SensorActive := Visu_L1.Door_2_SensorActive;

Visu_l1.Door_2_SensorOpen := IO_L1.Door_2_SensorOpen;
Visu_l1.Door_2_SensorClosed := IO_L1.Door_2_SensorClosed;
Visu_l1.Door_2_M_Open := IO_L1.Door_2_MotorOpen;
Visu_l1.Door_2_M_Close := IO_L1.Door_2_MotorClose;

fbL1_Door_3(
	MotorOpen:= IO_L1.Door_3_MotorOpen, 
	MotorClose:= IO_L1.Door_3_MotorClose,
	Position=> );
	
IO_L1.Door_3_SensorOpen := fbL1_Door_3.SensorOpenActive;
IO_L1.Door_3_SensorClosed := fbL1_Door_3.SensorCloseActive;
IO_L1.Door_3_SensorActive := Visu_L1.Door_3_SensorActive;

Visu_l1.Door_3_SensorOpen := IO_L1.Door_3_SensorOpen;
Visu_l1.Door_3_SensorClosed := IO_L1.Door_3_SensorClosed;
Visu_l1.Door_3_M_Open := IO_L1.Door_3_MotorOpen;
Visu_l1.Door_3_M_Close := IO_L1.Door_3_MotorClose;

fbL1_Door_4(
	MotorOpen:= IO_L1.Door_4_MotorOpen, 
	MotorClose:= IO_L1.Door_4_MotorClose,
	Position=> );
	
IO_L1.Door_4_SensorOpen := fbL1_Door_4.SensorOpenActive;
IO_L1.Door_4_SensorClosed := fbL1_Door_4.SensorCloseActive;
IO_L1.Door_4_SensorActive := Visu_L1.Door_4_SensorActive;

Visu_l1.Door_4_SensorOpen := IO_L1.Door_4_SensorOpen;
Visu_l1.Door_4_SensorClosed := IO_L1.Door_4_SensorClosed;
Visu_l1.Door_4_M_Open := IO_L1.Door_4_MotorOpen;
Visu_l1.Door_4_M_Close := IO_L1.Door_4_MotorClose;

fbL1_Door_5(
	MotorOpen:= IO_L1.Door_5_MotorOpen, 
	MotorClose:= IO_L1.Door_5_MotorClose,
	Position=> );
	
IO_L1.Door_5_SensorOpen := fbL1_Door_5.SensorOpenActive;
IO_L1.Door_5_SensorClosed := fbL1_Door_5.SensorCloseActive;
IO_L1.Door_5_SensorActive := Visu_L1.Door_5_SensorActive;

Visu_l1.Door_5_SensorOpen := IO_L1.Door_5_SensorOpen;
Visu_l1.Door_5_SensorClosed := IO_L1.Door_5_SensorClosed;
Visu_l1.Door_5_M_Open := IO_L1.Door_5_MotorOpen;
Visu_l1.Door_5_M_Close := IO_L1.Door_5_MotorClose;

fbL1_Door_6(
	MotorOpen:= IO_L1.Door_6_MotorOpen, 
	MotorClose:= IO_L1.Door_6_MotorClose,
	Position=> );
	
IO_L1.Door_6_SensorOpen := fbL1_Door_6.SensorOpenActive;
IO_L1.Door_6_SensorClosed := fbL1_Door_6.SensorCloseActive;
IO_L1.Door_6_SensorActive := Visu_L1.Door_6_SensorActive;

Visu_l1.Door_6_SensorOpen := IO_L1.Door_6_SensorOpen;
Visu_l1.Door_6_SensorClosed := IO_L1.Door_6_SensorClosed;
Visu_l1.Door_6_M_Open := IO_L1.Door_6_MotorOpen;
Visu_l1.Door_6_M_Close := IO_L1.Door_6_MotorClose;


// Update Visu

Visu_L1.Position_LIFT := fbL1_Axis.PositionInPercent;
Visu_L1.Door_1_Position := fbL1_Door_1.Position;
Visu_L1.Door_2_Position := fbL1_Door_2.Position;
Visu_L1.Door_3_Position := fbL1_Door_3.Position;
Visu_L1.Door_4_Position := fbL1_Door_4.Position;
Visu_L1.Door_5_Position := fbL1_Door_5.Position;
Visu_L1.Door_6_Position := fbL1_Door_6.Position;

Visu_L1.Panel_1_FloorNumber.0 := IO_L1.Panel_1_BCD_Bit[0];
Visu_L1.Panel_1_FloorNumber.1 := IO_L1.Panel_1_BCD_Bit[1];
Visu_L1.Panel_1_FloorNumber.2 := IO_L1.Panel_1_BCD_Bit[2];
Visu_L1.Panel_1_FloorNumber.3 := IO_L1.Panel_1_BCD_Bit[3];

Visu_L1.Panel_1_BtnLed := IO_L1.Panel_1_BtnLed;
Visu_L1.Panel_1_Led_Up := IO_L1.Panel_1_Led_Up;
Visu_L1.Panel_1_Led_Down := IO_L1.Panel_1_Led_Down;

IO_L1.Panel_1_Btn := Visu_L1.Panel_1_Btn;

Visu_L1.Panel_2_FloorNumber.0 := IO_L1.Panel_2_BCD_Bit[0];
Visu_L1.Panel_2_FloorNumber.1 := IO_L1.Panel_2_BCD_Bit[1];
Visu_L1.Panel_2_FloorNumber.2 := IO_L1.Panel_2_BCD_Bit[2];
Visu_L1.Panel_2_FloorNumber.3 := IO_L1.Panel_2_BCD_Bit[3];

Visu_L1.Panel_2_BtnLed := IO_L1.Panel_2_BtnLed;
Visu_L1.Panel_2_Led_Up := IO_L1.Panel_2_Led_Up;
Visu_L1.Panel_2_Led_Down := IO_L1.Panel_2_Led_Down;

IO_L1.Panel_2_Btn := Visu_L1.Panel_2_Btn;

Visu_L1.Panel_3_FloorNumber.0 := IO_L1.Panel_3_BCD_Bit[0];
Visu_L1.Panel_3_FloorNumber.1 := IO_L1.Panel_3_BCD_Bit[1];
Visu_L1.Panel_3_FloorNumber.2 := IO_L1.Panel_3_BCD_Bit[2];
Visu_L1.Panel_3_FloorNumber.3 := IO_L1.Panel_3_BCD_Bit[3];

Visu_L1.Panel_3_BtnLed := IO_L1.Panel_3_BtnLed;
Visu_L1.Panel_3_Led_Up := IO_L1.Panel_3_Led_Up;
Visu_L1.Panel_3_Led_Down := IO_L1.Panel_3_Led_Down;

IO_L1.Panel_3_Btn := Visu_L1.Panel_3_Btn;


Visu_L1.Panel_4_FloorNumber.0 := IO_L1.Panel_4_BCD_Bit[0];
Visu_L1.Panel_4_FloorNumber.1 := IO_L1.Panel_4_BCD_Bit[1];
Visu_L1.Panel_4_FloorNumber.2 := IO_L1.Panel_4_BCD_Bit[2];
Visu_L1.Panel_4_FloorNumber.3 := IO_L1.Panel_4_BCD_Bit[3];

Visu_L1.Panel_4_BtnLed := IO_L1.Panel_4_BtnLed;
Visu_L1.Panel_4_Led_Up := IO_L1.Panel_4_Led_Up;
Visu_L1.Panel_4_Led_Down := IO_L1.Panel_4_Led_Down;

IO_L1.Panel_4_Btn := Visu_L1.Panel_4_Btn;

Visu_L1.Panel_5_FloorNumber.0 := IO_L1.Panel_5_BCD_Bit[0];
Visu_L1.Panel_5_FloorNumber.1 := IO_L1.Panel_5_BCD_Bit[1];
Visu_L1.Panel_5_FloorNumber.2 := IO_L1.Panel_5_BCD_Bit[2];
Visu_L1.Panel_5_FloorNumber.3 := IO_L1.Panel_5_BCD_Bit[3];

Visu_L1.Panel_5_BtnLed := IO_L1.Panel_5_BtnLed;
Visu_L1.Panel_5_Led_Up := IO_L1.Panel_5_Led_Up;
Visu_L1.Panel_5_Led_Down := IO_L1.Panel_5_Led_Down;

IO_L1.Panel_5_Btn := Visu_L1.Panel_5_Btn;

Visu_L1.Panel_6_FloorNumber.0 := IO_L1.Panel_6_BCD_Bit[0];
Visu_L1.Panel_6_FloorNumber.1 := IO_L1.Panel_6_BCD_Bit[1];
Visu_L1.Panel_6_FloorNumber.2 := IO_L1.Panel_6_BCD_Bit[2];
Visu_L1.Panel_6_FloorNumber.3 := IO_L1.Panel_6_BCD_Bit[3];

Visu_L1.Panel_6_BtnLed := IO_L1.Panel_6_BtnLed;
Visu_L1.Panel_6_Led_Up := IO_L1.Panel_6_Led_Up;
Visu_L1.Panel_6_Led_Down := IO_L1.Panel_6_Led_Down;

IO_L1.Panel_6_Btn := Visu_L1.Panel_6_Btn;

Visu_L1.Control_LED_Blue := IO_L1.Control_LED_Blue;
Visu_L1.Control_LED_Red := IO_L1.Control_LED_Red;
Visu_L1.Control_LED_White := IO_L1.Control_LED_White;
Visu_L1.Control_LED_Yellow := IO_L1.Control_LED_Yellow;
IO_L1.Control_Start := Visu_L1.Control_Start;
IO_L1.Control_Reset := Visu_L1.Control_Reset;

IF Visu_L1.Control_State = 0 THEN
	IO_L1.Control_Automatic := FALSE;
	IO_L1.Control_Manual := FALSE;
ELSIF Visu_L1.Control_State = 1 THEN
	IO_L1.Control_Automatic := FALSE;
	IO_L1.Control_Manual := TRUE;
ELSIF Visu_L1.Control_State = 2 THEN
	IO_L1.Control_Automatic := TRUE;
	IO_L1.Control_Manual := FALSE;
END_IF

END_PROGRAM

// ---- 9_Modell/Lib/FB_MotionAxisPassive.TcPOU
FUNCTION_BLOCK FB_MotionAxisPassive
VAR_IN_OUT
	Axis : AXIS_REF;
END_VAR
VAR_INPUT
	RandomStart :BOOL := TRUE;
	Length : REAL := 1460.0;
	RefSensorPositionAbs : LREAL := 45;
	Window : LREAL := 5;
END_VAR
VAR_OUTPUT
	PositionInPercent : LREAL;
	CurrentPosition	: LREAL := Length / 2;
	RefSensor : BOOL;
	
END_VAR
VAR
	fbReadPosition : MC_ReadActualPosition;
	fbReadVelocity : MC_ReadActualVelocity;
	fbSetPosition : MC_SetPosition;
	fbReadStatus	: MC_ReadStatus;
	
	Random : DRAND;
	Initialize : BOOL := TRUE;
	SpeedStep : LREAL;
	RelStartPos : LREAL;
	LastPosition : LREAL;
	DeltaPosition: LREAL;
END_VAR


fbReadStatus(
	Axis:= Axis, 
	Enable:= TRUE);

IF Initialize THEN
	;
	Initialize := FALSE;
END_IF

fbSetPosition(
	Axis:= Axis, 
	Execute:= fbReadStatus.Valid, 
	Position:= 0);

IF fbReadStatus.Valid AND NOT fbSetPosition.Busy THEN		
	fbReadPosition(
		Axis:= Axis, 
		Enable:= TRUE);
		
	fbReadVelocity(
		Axis:= Axis, 
		Enable:= TRUE);
		
	DeltaPosition := fbReadPosition.Position - LastPosition;
	
	SpeedStep := F_SpeedPerCycle(fbReadVelocity.ActualVelocity);
	
	IF ABS(DeltaPosition) > 2 * ABS(SpeedStep) THEN
		DeltaPosition := 0;
	END_IF
	
	LastPosition := fbReadPosition.Position;	
	CurrentPosition := CurrentPosition + DeltaPosition;
END_IF

RefSensor :=  ((CurrentPosition > (RefSensorPositionAbs - Window)) AND (CurrentPosition < (RefSensorPositionAbs + Window)));

PositionInPercent := (100 * CurrentPosition) / LENGTH;

END_FUNCTION_BLOCK

// ---- 9_Modell/Lib/F_SpeedPerCycle.TcPOU
FUNCTION F_SpeedPerCycle : LREAL // Returns speed step per cycle [speed / cycle]
VAR_INPUT
	Speed : LREAL; // Speed in mm / s
END_VAR
VAR
	
END_VAR


F_SpeedPerCycle := Speed * UDINT_TO_LREAL(F_CycleTime()) / 1000.0;

END_FUNCTION

// ---- 9_Modell/Lib/F_CycleTime.TcPOU
FUNCTION F_CycleTime : UDINT // Returns current cycle time in [ms]
VAR_INPUT
END_VAR
VAR
	fbGetCurTaskIdx  : GETCURTASKINDEX;
END_VAR

fbGetCurTaskIdx();
F_CycleTime := _TaskInfo[fbGetCurTaskIdx.index].CycleTime / 10000;

END_FUNCTION

// ---- 9_Modell/Lib/FB_SimpleAxis.TcPOU
FUNCTION_BLOCK FB_SimpleAxis
(*
		Sensor 1					  Sensor 2
	  		|							|
	Left ----------------------------------- Right


*)
VAR_INPUT
	MotorOpen			: BOOL; // Motor turns right
	MotorClose			: BOOL; // Motor turns left
	Axis_Len			: REAL := 100; // Axis length [mm]
	SensorOpenOffset	: REAL := 6; // Sensor offset from left to sensor 1 position
	SensorCloseOffset	: REAL := 6; // Sensor offset from right to sensor 2 position
	StartPosition 		: REAL := Axis_Len / 2; // Start position axis
END_VAR
VAR_OUTPUT
	SensorOpenActive	: BOOL; // Sensor left is active
	SensorCloseActive	: BOOL; // Sensor right is active
	Position			: REAL := StartPosition; // Current axis position
END_VAR
VAR
	Step				: INT := 1; // Speed step
END_VAR


IF MotorOpen AND MotorClose THEN
	;
ELSIF MotorOpen THEN
	Position := Position + Step;
ELSIF MotorClose THEN
	Position := Position - Step;
END_IF

IF Position >= Axis_Len THEN
	Position := Axis_Len;
ELSIF Position <= 0 THEN
	Position := 0;
END_IF

SensorCloseActive := Position <= SensorCloseOffset;
SensorOpenActive := Position >= Axis_len - SensorOpenOffset;

END_FUNCTION_BLOCK

// ---- 0_App/MAIN.TcPOU
PROGRAM MAIN
VAR
	
	fbFahrleitsystem : FB_Fahrleitsystem;
	fbAchse : FB_Achse;
	fbManuell : FB_Manuell;
	fbTuer : FB_Tuer;
	fbTaskmanager : FB_Taskmanager_1;
	fbFahrlogikFIFO : FB_Logik_FIFO;
	fbFahrlogikShortestDistance : FB_Logik_ShortestDistance;
	fbPanel : FB_Panel ;
	LED_Loeschen_verstanden : BOOL;
	AutomatikmodusAktiv : BOOL;
	ManuellmodusAktiv : BOOL;
END_VAR

fbPanel(
    Panel_1_Btn := IO_L1.Panel_1_Btn,
    Panel_2_Btn := IO_L1.Panel_2_Btn,
    Panel_3_Btn := IO_L1.Panel_3_Btn,
    Panel_4_Btn := IO_L1.Panel_4_Btn,
    Panel_5_Btn := IO_L1.Panel_5_Btn,
    Panel_6_Btn := IO_L1.Panel_6_Btn,

    Panel_1_BtnLED => IO_L1.Panel_1_BtnLed,
    Panel_2_BtnLED => IO_L1.Panel_2_BtnLed,
    Panel_3_BtnLED => IO_L1.Panel_3_BtnLed,
    Panel_4_BtnLED => IO_L1.Panel_4_BtnLed,
    Panel_5_BtnLED => IO_L1.Panel_5_BtnLed,
    Panel_6_BtnLED => IO_L1.Panel_6_BtnLed,

    Panel_1_Led_Up => IO_L1.Panel_1_Led_Up,
    Panel_1_Led_Down => IO_L1.Panel_1_Led_Down,
    Panel_2_Led_Up => IO_L1.Panel_2_Led_Up,
    Panel_2_Led_Down => IO_L1.Panel_2_Led_Down,
    Panel_3_Led_Up => IO_L1.Panel_3_Led_Up,
    Panel_3_Led_Down => IO_L1.Panel_3_Led_Down,
    Panel_4_Led_Up => IO_L1.Panel_4_Led_Up,
    Panel_4_Led_Down => IO_L1.Panel_4_Led_Down,
    Panel_5_Led_Up => IO_L1.Panel_5_Led_Up,
    Panel_5_Led_Down => IO_L1.Panel_5_Led_Down,
    Panel_6_Led_Up => IO_L1.Panel_6_Led_Up,
    Panel_6_Led_Down => IO_L1.Panel_6_Led_Down,

    Panel_1_BCD_Bit => IO_L1.Panel_1_BCD_Bit,
    Panel_2_BCD_Bit => IO_L1.Panel_2_BCD_Bit,
    Panel_3_BCD_Bit => IO_L1.Panel_3_BCD_Bit,
    Panel_4_BCD_Bit => IO_L1.Panel_4_BCD_Bit,
    Panel_5_BCD_Bit => IO_L1.Panel_5_BCD_Bit,
    Panel_6_BCD_Bit => IO_L1.Panel_6_BCD_Bit,

    fbTaskManager := fbTaskmanager
);

fbTaskmanager(
    fbFahrleitsystem := fbFahrleitsystem,
    fbFahrlogik := fbFahrlogikFIFO
);

fbFahrleitsystem();

IF NOT fbFahrleitsystem.M_isBusy() AND IO_L1.Control_Manual THEN
	Divers.ManuellmodusAktiv := TRUE;
	Divers.AutomatikmodusAktiv := FALSE;
END_IF
IF IO_L1.Control_Automatic THEN
	Divers.AutomatikmodusAktiv := TRUE;
	Divers.ManuellmodusAktiv := FALSE;
END_IF

//LED Löschen
IF fbFahrleitsystem.M_AbholungFertig() > (-1) THEN
	LED_Loeschen_verstanden := fbPanel.M_TurnofLED(fbFahrleitsystem.M_AbholungFertig());
END_IF

fbManuell();

END_PROGRAM

// ---- 0_App/Lib/FB_Fahrleitsystem.TcPOU
FUNCTION_BLOCK FB_Fahrleitsystem
VAR_INPUT
END_VAR
VAR_OUTPUT
END_VAR
VAR
	Done : BOOL;
	Busy	: BOOL;
	Error : BOOL;
	StartStockwerk:	INT;
	ZielStockwerk:	INT;
	SicherheitsCheckbestanden : BOOL;
	AmStartStockwerk : BOOL;
	AmZielStockwerk : BOOL;
	TuerenZu : BOOL;
	Start : BOOL;
	AktuellesStockwerk : INT;
	Fahrauftragverstanden : BOOL;
	Tuerauftragverstanden : BOOL;
	State: ENUM_Fahrsystem;
	fbTuer : FB_Tuer;
	fbAchse : FB_Achse;
	AbholungFertig : BOOL;
	Closingdoors: BOOL;
	Achsereferenziert: BOOL;
	AufstartenAbgeschlossen : BOOL;
	AufstartenFreigabe : BOOL;
	AllDoorsClosed : BOOL;
	fbBlinker : FB_Blinker;
	FehlerQuittierenFlanke : R_TRIG;   // NEU — Flanke für Quittierung
 	sFehlertext : STRING(500);  // lokale Hilfsvariable
    i_txt       : INT;
END_VAR

fbAchse(Simulation:= , S_Zielposition:= , Achse:= IO_L1.LiftAxis);
fbTuer(
    SensorOpen1 := IO_L1.Door_1_SensorOpen,
    SensorOpen2 := IO_L1.Door_2_SensorOpen,
    SensorOpen3 := IO_L1.Door_3_SensorOpen,
    SensorOpen4 := IO_L1.Door_4_SensorOpen,
    SensorOpen5 := IO_L1.Door_5_SensorOpen,
    SensorOpen6 := IO_L1.Door_6_SensorOpen,

    SensorClosed1 := IO_L1.Door_1_SensorClosed,
    SensorClosed2 := IO_L1.Door_2_SensorClosed,
    SensorClosed3 := IO_L1.Door_3_SensorClosed,
    SensorClosed4 := IO_L1.Door_4_SensorClosed,
    SensorClosed5 := IO_L1.Door_5_SensorClosed,
    SensorClosed6 := IO_L1.Door_6_SensorClosed,

    Lichtschranke1 := IO_L1.Door_1_SensorActive,
    Lichtschranke2 := IO_L1.Door_2_SensorActive,
    Lichtschranke3 := IO_L1.Door_3_SensorActive,
    Lichtschranke4 := IO_L1.Door_4_SensorActive,
    Lichtschranke5 := IO_L1.Door_5_SensorActive,
    Lichtschranke6 := IO_L1.Door_6_SensorActive,

    MotorOpen1 => IO_L1.Door_1_MotorOpen,
    MotorOpen2 => IO_L1.Door_2_MotorOpen,
    MotorOpen3 => IO_L1.Door_3_MotorOpen,
    MotorOpen4 => IO_L1.Door_4_MotorOpen,
    MotorOpen5 => IO_L1.Door_5_MotorOpen,
    MotorOpen6 => IO_L1.Door_6_MotorOpen,

    MotorClose1 => IO_L1.Door_1_MotorClose,
    MotorClose2 => IO_L1.Door_2_MotorClose,
    MotorClose3 => IO_L1.Door_3_MotorClose,
    MotorClose4 => IO_L1.Door_4_MotorClose,
    MotorClose5 => IO_L1.Door_5_MotorClose,
    MotorClose6 => IO_L1.Door_6_MotorClose,
	AllDoorsClosed => AllDoorsClosed,
	FehlerQuittieren := IO_L1.Control_Reset
);

fbBlinker(bEnable:= TRUE, tOn:= T#500MS, tOff:=T#500MS , bOut=> );
SicherheitsCheckbestanden := FALSE;
Done := FALSE;
CASE State OF


	ENUM_Fahrsystem.Warten:
		Busy := FALSE;
		Done := FALSE;
		IF NOT 	AufstartenAbgeschlossen  AND IO_L1.Control_Automatic THEN
			Busy := TRUE;
			State := ENUM_Fahrsystem.Aufstartablauf;
		END_IF
		IF Start AND Divers.AutomatikmodusAktiv THEN
			Busy := TRUE;
			Start := FALSE;
			State := ENUM_Fahrsystem.Sicherheitscheck;
		END_IF
 		IF Visu_Manuellmodus.PosAnfahren AND Divers.ManuellmodusAktiv THEN
			ZielStockwerk := Visu_Manuellmodus.Zielstock;
 			State := ENUM_Fahrsystem.ZumZielStockwerk; 
		END_IF
	ENUM_Fahrsystem.Sicherheitscheck:
		//IF fbTuer.M_AreDoorsClosed() AND NOT fbAchse.M_isBusy() AND NOT fbAchse.M_hasError() THEN
			SicherheitsCheckbestanden := TRUE;
		//END_IF
		IF SicherheitsCheckbestanden THEN
			IF StartStockwerk = AktuellesStockwerk THEN
				State := ENUM_Fahrsystem.ZumZielStockwerk;
			END_IF
			IF StartStockwerk <> AktuellesStockwerk THEN 
				State := ENUM_Fahrsystem.ZumStartStockwerk;
			END_IF
		END_IF
		
	ENUM_Fahrsystem.Tueren:
		Busy := TRUE;	
		IF NOT Tuerauftragverstanden AND NOT fbAchse.M_isBusy() AND NOT fbAchse.M_hasError()THEN
			Tuerauftragverstanden := fbTuer.M_Tuerablaufstarten(AktuellesStockwerk);
		END_IF
		IF fbTuer.M_DoorOpen() THEN
			AbholungFertig := TRUE;
		ELSE 
			AbholungFertig := FALSE;
		END_IF
		IF fbTuer.M_isDone() THEN
			AbholungFertig := FALSE;
			Tuerauftragverstanden := FALSE;
			IF AmStartStockwerk THEN
				State := ENUM_Fahrsystem.ZumZielStockwerk;
			END_IF
			IF AmZielStockwerk THEN
				Done := TRUE; 
				State := ENUM_Fahrsystem.Warten;
			END_IF
		END_IF
	ENUM_Fahrsystem.ZumStartStockwerk:
		Busy := TRUE;
		AmZielStockwerk := FALSE;
		Fahrauftragverstanden := fbAchse.M_Movetoposition(StartStockwerk);
		IF fbAchse.M_isDone() THEN
			//OrderID_Counter.AktuellesStockwerk := StartStockwerk;
			AktuellesStockwerk := StartStockwerk;
			AmStartStockwerk := TRUE;
			State := ENUM_Fahrsystem.Tueren;
		END_IF
	ENUM_Fahrsystem.ZumZielStockwerk:
		Busy := TRUE;
		AmStartStockwerk := FALSE;
		Fahrauftragverstanden := fbAchse.M_Movetoposition(ZielStockwerk);
		IF fbAchse.M_isDone() THEN
			//OrderID_Counter.AktuellesStockwerk := ZielStockwerk;
			AktuellesStockwerk := ZielStockwerk;
			AmZielStockwerk := TRUE;
			IF Divers.AutomatikmodusAktiv THEN
				State := ENUM_Fahrsystem.Tueren;
			ELSE
				State := ENUM_Fahrsystem.Warten;	
			END_IF
			
		END_IF
	
	ENUM_Fahrsystem.Aufstartablauf: 
	Busy := TRUE;
	IF IO_L1.Control_Start THEN
		AufstartenFreigabe := TRUE;
	END_IF
		IF AufstartenFreigabe THEN
	
			IF NOT AllDoorsClosed THEN
				IO_L1.Control_LED_White := TRUE;
				Closingdoors := fbTuer.M_closeAllDoors();
			END_IF
			IF AllDoorsClosed THEN
				IO_L1.Control_LED_Red := TRUE;
				Achsereferenziert := fbAchse.M_Movetoposition(1);
					IF fbAchse.M_isDone() THEN
						AktuellesStockwerk := 1;
						AufstartenAbgeschlossen := TRUE;
						AufstartenFreigabe := FALSE;
						State := ENUM_Fahrsystem.Warten;
				END_IF
			END_IF
			
		END_IF
		
END_CASE


//LED Stuerung
IF IO_L1.Control_Automatic AND AufstartenAbgeschlossen THEN
    // Anlage läuft (mit oder ohne Auftrag) → dauernd an
    IO_L1.Control_LED_White := TRUE;

ELSIF IO_L1.Control_Automatic AND NOT AufstartenAbgeschlossen THEN
    // Aufstartablauf → blinken
    IO_L1.Control_LED_White := fbBlinker.bOut;

ELSIF NOT IO_L1.Control_Automatic AND Busy THEN
    // Automatik verlassen, Auftrag wird noch fertig gemacht → blinken
    IO_L1.Control_LED_White := fbBlinker.bOut;

ELSE
    // Kein Automatik, kein aktiver Auftrag → aus
    IO_L1.Control_LED_White := FALSE;
END_IF
// ── Fehler sammeln ────────────────────────────────────────────────────────────
Divers.Fehler.AchsePower := fbAchse.fbPower.Error;
Divers.Fehler.AchseHome  := fbAchse.fbHome.Error;
Divers.Fehler.AchseMove  := fbAchse.fbMoveAbs.Error;
Divers.Fehler.AchseJog   := fbAchse.fbJog.Error;
Divers.Fehler.NotAus     := IO_L1.Control_EmergencyStopActive;
Divers.Fehler.TuerTimeout := fbTuer.TuerFehler;

// Letzten Achsen-Fehlercode speichern
IF fbAchse.fbPower.Error   THEN Divers.Fehler.AchseFehlercode := fbAchse.FehlercodePower; END_IF
IF fbAchse.fbHome.Error    THEN Divers.Fehler.AchseFehlercode := fbAchse.FehlercodeRef;   END_IF
IF fbAchse.fbMoveAbs.Error THEN Divers.Fehler.AchseFehlercode := fbAchse.FehlercodeMove;  END_IF

// Zusammenfassung
Divers.Fehler.IrgendeinFehler :=
    Divers.Fehler.AchsePower OR
    Divers.Fehler.AchseHome  OR
    Divers.Fehler.AchseMove  OR
    Divers.Fehler.AchseJog   OR
    Divers.Fehler.NotAus     OR
    Divers.Fehler.TuerTimeout[1] OR Divers.Fehler.TuerTimeout[2] OR
    Divers.Fehler.TuerTimeout[3] OR Divers.Fehler.TuerTimeout[4] OR
    Divers.Fehler.TuerTimeout[5] OR Divers.Fehler.TuerTimeout[6];

Divers.Fehler.IrgendEineWarnung := IO_L1.Control_Overload;

// ── Quittierung ───────────────────────────────────────────────────────────────
FehlerQuittierenFlanke(CLK := IO_L1.Control_Reset);
IF FehlerQuittierenFlanke.Q AND NOT Divers.Fehler.IrgendeinFehler THEN
    Divers.Fehler.FehlerQuittiert := TRUE;
END_IF
IF Divers.Fehler.IrgendeinFehler THEN
    Divers.Fehler.FehlerQuittiert := FALSE;  // Reset bei neuem Fehler
END_IF

// ── LED Steuerung Rot / Blau / Gelb ──────────────────────────────────────────
IF Divers.Fehler.IrgendeinFehler THEN
    IO_L1.Control_LED_Red := TRUE;
    IF Divers.Fehler.FehlerQuittiert THEN
        IO_L1.Control_LED_Blue := fbBlinker.bOut;  // blinkt = quittierbar
    ELSE
        IO_L1.Control_LED_Blue := TRUE;             // dauernd = noch aktiv
    END_IF
ELSE
    IO_L1.Control_LED_Red  := FALSE;
    IO_L1.Control_LED_Blue := FALSE;
END_IF

IO_L1.Control_LED_Yellow := Divers.Fehler.IrgendEineWarnung;
// ─────────────────────────────────────────────────────────────────────────────
// ── Fehlertext aufbauen ───────────────────────────────────────────────────────
sFehlertext := '';

// Achse
IF Divers.Fehler.AchsePower THEN
    sFehlertext := CONCAT(sFehlertext, 'FEHLER: Achse Power');
    sFehlertext := CONCAT(sFehlertext, CONCAT(' (Code: ', CONCAT(UDINT_TO_STRING(Divers.Fehler.AchseFehlercode), ') | ')));
END_IF
IF Divers.Fehler.AchseHome THEN
    sFehlertext := CONCAT(sFehlertext, 'FEHLER: Referenzfahrt');
    sFehlertext := CONCAT(sFehlertext, CONCAT(' (Code: ', CONCAT(UDINT_TO_STRING(Divers.Fehler.AchseFehlercode), ') | ')));
END_IF
IF Divers.Fehler.AchseMove THEN
    sFehlertext := CONCAT(sFehlertext, 'FEHLER: Positionierung');
    sFehlertext := CONCAT(sFehlertext, CONCAT(' (Code: ', CONCAT(UDINT_TO_STRING(Divers.Fehler.AchseFehlercode), ') | ')));
END_IF
IF Divers.Fehler.AchseJog THEN
    sFehlertext := CONCAT(sFehlertext, 'FEHLER: Jog | ');
END_IF

// Türen
FOR i_txt := 1 TO 6 DO
    IF Divers.Fehler.TuerTimeout[i_txt] THEN
        sFehlertext := CONCAT(sFehlertext, 'FEHLER: Tuer Timeout Stock. ');
        sFehlertext := CONCAT(sFehlertext, CONCAT(INT_TO_STRING(i_txt), ' | '));
    END_IF
END_FOR

// Allgemein
IF Divers.Fehler.NotAus THEN
    sFehlertext := CONCAT(sFehlertext, 'FEHLER: Not-Aus | ');
END_IF
IF Divers.Fehler.Brandalarm THEN
    sFehlertext := CONCAT(sFehlertext, 'FEHLER: Brandalarm | ');
END_IF

// Warnung
IF Divers.Fehler.IrgendEineWarnung THEN
    sFehlertext := CONCAT(sFehlertext, 'WARNUNG: Ueberlast Kabine | ');
END_IF

// Kein Fehler
IF sFehlertext = '' THEN
    sFehlertext := 'Keine Fehler';
END_IF

Divers.Fehlertext := sFehlertext;
// ─────────────────────────────────────────────────────────────────────────────

METHOD PUBLIC M_AbholungFertig : INT
VAR_INPUT
END_VAR
IF AbholungFertig THEN
	M_AbholungFertig := ZielStockwerk;
ELSE
	M_AbholungFertig := -1;
END_IF
END_METHOD

METHOD PUBLIC M_AcceptTask : BOOL
VAR_INPUT
Task : ST_Fahrauftrag;

END_VAR
IF NOT Busy THEN
	StartStockwerk := Task.Startstockwerk;
	Zielstockwerk := Task.Zielstockwerk;
	Start:= TRUE;
	M_AcceptTask := TRUE;
ELSE 
	M_AcceptTask := FALSE;
END_IF
END_METHOD

METHOD PUBLIC M_isBusy : BOOL
VAR_INPUT
END_VAR
M_isBusy := Busy;
END_METHOD

METHOD PUBLIC M_isDone : BOOL
VAR_INPUT
END_VAR
M_isDone := Done;
END_METHOD

END_FUNCTION_BLOCK

// ---- 0_App/Lib/FB_Tuer.TcPOU
FUNCTION_BLOCK FB_Tuer
VAR_INPUT
	SensorOpen1 : BOOL;
	SensorOpen2 : BOOL;
	SensorOpen3 : BOOL;
	SensorOpen4 : BOOL;
	SensorOpen5 : BOOL;
	SensorOpen6 : BOOL;
	
	SensorClosed1 : BOOL;
	SensorClosed2 : BOOL;
	SensorClosed3 : BOOL;
	SensorClosed4 : BOOL;
	SensorClosed5 : BOOL;
	SensorClosed6 : BOOL;
	
	Lichtschranke1 : BOOL;
	Lichtschranke2 : BOOL;
	Lichtschranke3 : BOOL;
	Lichtschranke4 : BOOL;
	Lichtschranke5 : BOOL;
	Lichtschranke6 : BOOL;
	FehlerQuittieren : BOOL;   // NEU — von FB_Fahrleitsystem gesetzt
END_VAR
VAR_OUTPUT
	MotorOpen1 : BOOL;
	MotorOpen2 : BOOL;
	MotorOpen3 : BOOL;
	MotorOpen4 : BOOL;
	MotorOpen5 : BOOL;
	MotorOpen6 : BOOL;
	
	MotorClose1 : BOOL;
	MotorClose2 : BOOL;
	MotorClose3 : BOOL;
	MotorClose4 : BOOL;
	MotorClose5 : BOOL;
	MotorClose6 : BOOL;
	Done : BOOL;
	AllDoorsClosed : BOOL;
END_VAR
VAR
	TuerzyklusStarten : BOOL;
	Stockwerk : INT;
	State : ENUM_Tuer;
	ton1 : TON;
	ton2 : TON;
	ton3 : TON;
	ton4 : TON;
	ton5 : TON;
	ton6 : TON;
	Tueroffen : BOOL;
	bCloseAllMode : BOOL;
	tonOpenTimeout  : ARRAY[1..6] OF TON;   // NEU
	tonCloseTimeout : ARRAY[1..6] OF TON;   // NEU
	TuerFehler      : ARRAY[1..6] OF BOOL;  // NEU — Output für Fehlersammlung
	i_err           : INT;                  // NEU — Laufvariable
END_VAR

// ── Tür Timeout Überwachung ──────────────────────────────────────────────────
tonOpenTimeout[1](IN := MotorOpen1 AND NOT SensorOpen1, PT := T#3S);
tonOpenTimeout[2](IN := MotorOpen2 AND NOT SensorOpen2, PT := T#3S);
tonOpenTimeout[3](IN := MotorOpen3 AND NOT SensorOpen3, PT := T#3S);
tonOpenTimeout[4](IN := MotorOpen4 AND NOT SensorOpen4, PT := T#3S);
tonOpenTimeout[5](IN := MotorOpen5 AND NOT SensorOpen5, PT := T#3S);
tonOpenTimeout[6](IN := MotorOpen6 AND NOT SensorOpen6, PT := T#3S);

tonCloseTimeout[1](IN := MotorClose1 AND NOT SensorClosed1, PT := T#3S);
tonCloseTimeout[2](IN := MotorClose2 AND NOT SensorClosed2, PT := T#3S);
tonCloseTimeout[3](IN := MotorClose3 AND NOT SensorClosed3, PT := T#3S);
tonCloseTimeout[4](IN := MotorClose4 AND NOT SensorClosed4, PT := T#3S);
tonCloseTimeout[5](IN := MotorClose5 AND NOT SensorClosed5, PT := T#3S);
tonCloseTimeout[6](IN := MotorClose6 AND NOT SensorClosed6, PT := T#3S);

// Fehler setzen bei Timeout
FOR i_err := 1 TO 6 DO
    IF tonOpenTimeout[i_err].Q OR tonCloseTimeout[i_err].Q THEN
        TuerFehler[i_err] := TRUE;
    END_IF
END_FOR

// Motoren sofort stoppen bei Türfehler
IF TuerFehler[1] THEN MotorOpen1 := FALSE; MotorClose1 := FALSE; END_IF
IF TuerFehler[2] THEN MotorOpen2 := FALSE; MotorClose2 := FALSE; END_IF
IF TuerFehler[3] THEN MotorOpen3 := FALSE; MotorClose3 := FALSE; END_IF
IF TuerFehler[4] THEN MotorOpen4 := FALSE; MotorClose4 := FALSE; END_IF
IF TuerFehler[5] THEN MotorOpen5 := FALSE; MotorClose5 := FALSE; END_IF
IF TuerFehler[6] THEN MotorOpen6 := FALSE; MotorClose6 := FALSE; END_IF

// Quittierung
IF FehlerQuittieren THEN
    FOR i_err := 1 TO 6 DO
        TuerFehler[i_err] := FALSE;
    END_FOR
END_IF
// ────────────────────────────────────────────────────────────────────────────

Done := FALSE;

// AllDoorsClosed immer prüfen – unabhängig vom Modus
IF IO_L1.Door_1_SensorClosed AND IO_L1.Door_2_SensorClosed AND IO_L1.Door_3_SensorClosed
   AND IO_L1.Door_4_SensorClosed AND IO_L1.Door_5_SensorClosed AND IO_L1.Door_6_SensorClosed THEN
    AllDoorsClosed := TRUE;
	Divers.AlleTuerenZu := TRUE;
ELSE
	Divers.AlleTuerenZu := FALSE;
    AllDoorsClosed := FALSE;
END_IF

// ── AUTOMATIK ────────────────────────────────────────────────────────────────
IF Divers.AutomatikmodusAktiv THEN

    ton1(IN := State = ENUM_Tuer.TuereAuf AND SensorOpen1, PT := T#2S);
    ton2(IN := State = ENUM_Tuer.TuereAuf AND SensorOpen2, PT := T#2S);
    ton3(IN := State = ENUM_Tuer.TuereAuf AND SensorOpen3, PT := T#2S);
    ton4(IN := State = ENUM_Tuer.TuereAuf AND SensorOpen4, PT := T#2S);
    ton5(IN := State = ENUM_Tuer.TuereAuf AND SensorOpen5, PT := T#2S);
    ton6(IN := State = ENUM_Tuer.TuereAuf AND SensorOpen6, PT := T#2S);

    IF bCloseAllMode THEN
        MotorOpen1 := FALSE;
        IF NOT Lichtschranke1 THEN
            MotorClose1 := FALSE;
        ELSIF NOT SensorClosed1 THEN
            MotorClose1 := TRUE;
        ELSE
            MotorClose1 := FALSE;
        END_IF
        MotorOpen2 := FALSE;
        IF NOT Lichtschranke2 THEN
            MotorClose2 := FALSE;
        ELSIF NOT SensorClosed2 THEN
            MotorClose2 := TRUE;
        ELSE
            MotorClose2 := FALSE;
        END_IF
        MotorOpen3 := FALSE;
        IF NOT Lichtschranke3 THEN
            MotorClose3 := FALSE;
        ELSIF NOT SensorClosed3 THEN
            MotorClose3 := TRUE;
        ELSE
            MotorClose3 := FALSE;
        END_IF
        MotorOpen4 := FALSE;
        IF NOT Lichtschranke4 THEN
            MotorClose4 := FALSE;
        ELSIF NOT SensorClosed4 THEN
            MotorClose4 := TRUE;
        ELSE
            MotorClose4 := FALSE;
        END_IF
        MotorOpen5 := FALSE;
        IF NOT Lichtschranke5 THEN
            MotorClose5 := FALSE;
        ELSIF NOT SensorClosed5 THEN
            MotorClose5 := TRUE;
        ELSE
            MotorClose5 := FALSE;
        END_IF
        MotorOpen6 := FALSE;
        IF NOT Lichtschranke6 THEN
            MotorClose6 := FALSE;
        ELSIF NOT SensorClosed6 THEN
            MotorClose6 := TRUE;
        ELSE
            MotorClose6 := FALSE;
        END_IF
        IF SensorClosed1 AND SensorClosed2 AND SensorClosed3
           AND SensorClosed4 AND SensorClosed5 AND SensorClosed6 THEN
            bCloseAllMode := FALSE;
            Done := TRUE;
        END_IF
    ELSE
        MotorOpen1 := FALSE; MotorClose1 := FALSE;
        MotorOpen2 := FALSE; MotorClose2 := FALSE;
        MotorOpen3 := FALSE; MotorClose3 := FALSE;
        MotorOpen4 := FALSE; MotorClose4 := FALSE;
        MotorOpen5 := FALSE; MotorClose5 := FALSE;
        MotorOpen6 := FALSE; MotorClose6 := FALSE;
        CASE State OF
            ENUM_Tuer.TuereZu:
                IF TuerzyklusStarten AND Stockwerk = 1 THEN State := ENUM_Tuer.TuereOeffnen; END_IF
                IF TuerzyklusStarten AND Stockwerk = 2 THEN State := ENUM_Tuer.TuereOeffnen; END_IF
                IF TuerzyklusStarten AND Stockwerk = 3 THEN State := ENUM_Tuer.TuereOeffnen; END_IF
                IF TuerzyklusStarten AND Stockwerk = 4 THEN State := ENUM_Tuer.TuereOeffnen; END_IF
                IF TuerzyklusStarten AND Stockwerk = 5 THEN State := ENUM_Tuer.TuereOeffnen; END_IF
                IF TuerzyklusStarten AND Stockwerk = 6 THEN State := ENUM_Tuer.TuereOeffnen; END_IF
            ENUM_Tuer.TuereOeffnen:
                Tueroffen := TRUE;
                IF Stockwerk = 1 THEN
                    IF NOT SensorOpen1 THEN MotorOpen1 := TRUE;
                    ELSE MotorOpen1 := FALSE; State := ENUM_Tuer.TuereAuf; END_IF
                END_IF
                IF Stockwerk = 2 THEN
                    IF NOT SensorOpen2 THEN MotorOpen2 := TRUE;
                    ELSE MotorOpen2 := FALSE; State := ENUM_Tuer.TuereAuf; END_IF
                END_IF
                IF Stockwerk = 3 THEN
                    IF NOT SensorOpen3 THEN MotorOpen3 := TRUE;
                    ELSE MotorOpen3 := FALSE; State := ENUM_Tuer.TuereAuf; END_IF
                END_IF
                IF Stockwerk = 4 THEN
                    IF NOT SensorOpen4 THEN MotorOpen4 := TRUE;
                    ELSE MotorOpen4 := FALSE; State := ENUM_Tuer.TuereAuf; END_IF
                END_IF
                IF Stockwerk = 5 THEN
                    IF NOT SensorOpen5 THEN MotorOpen5 := TRUE;
                    ELSE MotorOpen5 := FALSE; State := ENUM_Tuer.TuereAuf; END_IF
                END_IF
                IF Stockwerk = 6 THEN
                    IF NOT SensorOpen6 THEN MotorOpen6 := TRUE;
                    ELSE MotorOpen6 := FALSE; State := ENUM_Tuer.TuereAuf; END_IF
                END_IF
            ENUM_Tuer.TuereAuf:
                Tueroffen := FALSE;
                IF Stockwerk = 1 AND ton1.Q THEN State := ENUM_Tuer.TuereSchliessen; END_IF
                IF Stockwerk = 2 AND ton2.Q THEN State := ENUM_Tuer.TuereSchliessen; END_IF
                IF Stockwerk = 3 AND ton3.Q THEN State := ENUM_Tuer.TuereSchliessen; END_IF
                IF Stockwerk = 4 AND ton4.Q THEN State := ENUM_Tuer.TuereSchliessen; END_IF
                IF Stockwerk = 5 AND ton5.Q THEN State := ENUM_Tuer.TuereSchliessen; END_IF
                IF Stockwerk = 6 AND ton6.Q THEN State := ENUM_Tuer.TuereSchliessen; END_IF
            ENUM_Tuer.TuereSchliessen:
                IF Stockwerk = 1 THEN
                    IF NOT Lichtschranke1 THEN MotorClose1 := FALSE; State := ENUM_Tuer.TuereOeffnen;
                    ELSIF NOT SensorClosed1 THEN MotorClose1 := TRUE;
                    ELSE MotorClose1 := FALSE; TuerzyklusStarten := FALSE; Done := TRUE; State := ENUM_Tuer.TuereZu; END_IF
                END_IF
                IF Stockwerk = 2 THEN
                    IF NOT Lichtschranke2 THEN MotorClose2 := FALSE; State := ENUM_Tuer.TuereOeffnen;
                    ELSIF NOT SensorClosed2 THEN MotorClose2 := TRUE;
                    ELSE MotorClose2 := FALSE; TuerzyklusStarten := FALSE; Done := TRUE; State := ENUM_Tuer.TuereZu; END_IF
                END_IF
                IF Stockwerk = 3 THEN
                    IF NOT Lichtschranke3 THEN MotorClose3 := FALSE; State := ENUM_Tuer.TuereOeffnen;
                    ELSIF NOT SensorClosed3 THEN MotorClose3 := TRUE;
                    ELSE MotorClose3 := FALSE; TuerzyklusStarten := FALSE; Done := TRUE; State := ENUM_Tuer.TuereZu; END_IF
                END_IF
                IF Stockwerk = 4 THEN
                    IF NOT Lichtschranke4 THEN MotorClose4 := FALSE; State := ENUM_Tuer.TuereOeffnen;
                    ELSIF NOT SensorClosed4 THEN MotorClose4 := TRUE;
                    ELSE MotorClose4 := FALSE; TuerzyklusStarten := FALSE; Done := TRUE; State := ENUM_Tuer.TuereZu; END_IF
                END_IF
                IF Stockwerk = 5 THEN
                    IF NOT Lichtschranke5 THEN MotorClose5 := FALSE; State := ENUM_Tuer.TuereOeffnen;
                    ELSIF NOT SensorClosed5 THEN MotorClose5 := TRUE;
                    ELSE MotorClose5 := FALSE; TuerzyklusStarten := FALSE; Done := TRUE; State := ENUM_Tuer.TuereZu; END_IF
                END_IF
                IF Stockwerk = 6 THEN
                    IF NOT Lichtschranke6 THEN MotorClose6 := FALSE; State := ENUM_Tuer.TuereOeffnen;
                    ELSIF NOT SensorClosed6 THEN MotorClose6 := TRUE;
                    ELSE MotorClose6 := FALSE; TuerzyklusStarten := FALSE; Done := TRUE; State := ENUM_Tuer.TuereZu; END_IF
                END_IF
            ENUM_Tuer.Error:
        END_CASE
    END_IF

// ── MANUELL ──────────────────────────────────────────────────────────────────
ELSIF Divers.ManuellmodusAktiv THEN

    // Alle Ausgänge zuerst zurücksetzen
    MotorOpen1 := FALSE; MotorClose1 := FALSE;
    MotorOpen2 := FALSE; MotorClose2 := FALSE;
    MotorOpen3 := FALSE; MotorClose3 := FALSE;
    MotorOpen4 := FALSE; MotorClose4 := FALSE;
    MotorOpen5 := FALSE; MotorClose5 := FALSE;
    MotorOpen6 := FALSE; MotorClose6 := FALSE;

    // Einzelne Türen – Auf
    IF Visu_Manuellmodus.bTuerAuf[1] AND NOT SensorOpen1 THEN MotorOpen1 := TRUE; END_IF
    IF Visu_Manuellmodus.bTuerAuf[2] AND NOT SensorOpen2 THEN MotorOpen2 := TRUE; END_IF
    IF Visu_Manuellmodus.bTuerAuf[3] AND NOT SensorOpen3 THEN MotorOpen3 := TRUE; END_IF
    IF Visu_Manuellmodus.bTuerAuf[4] AND NOT SensorOpen4 THEN MotorOpen4 := TRUE; END_IF
    IF Visu_Manuellmodus.bTuerAuf[5] AND NOT SensorOpen5 THEN MotorOpen5 := TRUE; END_IF
    IF Visu_Manuellmodus.bTuerAuf[6] AND NOT SensorOpen6 THEN MotorOpen6 := TRUE; END_IF

    // Einzelne Türen – Zu (Lichtschranke beachten)
    IF Visu_Manuellmodus.bTuerZu[1] AND NOT SensorClosed1 AND Lichtschranke1 THEN MotorClose1 := TRUE; END_IF
    IF Visu_Manuellmodus.bTuerZu[2] AND NOT SensorClosed2 AND Lichtschranke2 THEN MotorClose2 := TRUE; END_IF
    IF Visu_Manuellmodus.bTuerZu[3] AND NOT SensorClosed3 AND Lichtschranke3 THEN MotorClose3 := TRUE; END_IF
    IF Visu_Manuellmodus.bTuerZu[4] AND NOT SensorClosed4 AND Lichtschranke4 THEN MotorClose4 := TRUE; END_IF
    IF Visu_Manuellmodus.bTuerZu[5] AND NOT SensorClosed5 AND Lichtschranke5 THEN MotorClose5 := TRUE; END_IF
    IF Visu_Manuellmodus.bTuerZu[6] AND NOT SensorClosed6 AND Lichtschranke6 THEN MotorClose6 := TRUE; END_IF

    // Alle Türen auf
    IF Visu_Manuellmodus.AlleTuerenAuf THEN
        IF NOT SensorOpen1 THEN MotorOpen1 := TRUE; END_IF
        IF NOT SensorOpen2 THEN MotorOpen2 := TRUE; END_IF
        IF NOT SensorOpen3 THEN MotorOpen3 := TRUE; END_IF
        IF NOT SensorOpen4 THEN MotorOpen4 := TRUE; END_IF
        IF NOT SensorOpen5 THEN MotorOpen5 := TRUE; END_IF
        IF NOT SensorOpen6 THEN MotorOpen6 := TRUE; END_IF
    END_IF

    // Alle Türen zu (Lichtschranke beachten)
    IF Visu_Manuellmodus.AlleTuerenZu THEN
        IF NOT SensorClosed1 AND Lichtschranke1 THEN MotorClose1 := TRUE; END_IF
        IF NOT SensorClosed2 AND Lichtschranke2 THEN MotorClose2 := TRUE; END_IF
        IF NOT SensorClosed3 AND Lichtschranke3 THEN MotorClose3 := TRUE; END_IF
        IF NOT SensorClosed4 AND Lichtschranke4 THEN MotorClose4 := TRUE; END_IF
        IF NOT SensorClosed5 AND Lichtschranke5 THEN MotorClose5 := TRUE; END_IF
        IF NOT SensorClosed6 AND Lichtschranke6 THEN MotorClose6 := TRUE; END_IF
    END_IF

END_IF

METHOD PUBLIC M_AreDoorsClosed : BOOL
VAR_INPUT
END_VAR
IF IO_L1.Door_1_SensorClosed AND IO_L1.Door_2_SensorClosed AND IO_L1.Door_3_SensorClosed AND IO_L1.Door_4_SensorClosed AND IO_L1.Door_5_SensorClosed AND IO_L1.Door_6_SensorClosed THEN
	M_AreDoorsClosed := TRUE;
ELSE
	M_AreDoorsClosed := FALSE;
END_IF
END_METHOD

METHOD PUBLIC M_closeAllDoors : BOOL
VAR_INPUT
END_VAR
VAR
	Tuer1zu : BOOL;
	Tuer2zu : BOOL;
	Tuer3zu : BOOL;
	Tuer4zu : BOOL;
	Tuer5zu : BOOL;
	Tuer6zu : BOOL;
END_VAR

bCloseAllMode := TRUE;

M_closeAllDoors :=
    SensorClosed1 AND SensorClosed2 AND SensorClosed3 AND
    SensorClosed4 AND SensorClosed5 AND SensorClosed6;
END_METHOD

METHOD PUBLIC M_DoorOpen : BOOL
VAR_INPUT
	
END_VAR
IF Tueroffen THEN
	M_DoorOpen := TRUE;
ELSE
	M_DoorOpen := FALSE;
END_IF
END_METHOD

METHOD PUBLIC M_isDone : BOOL
VAR_INPUT
END_VAR
IF Done THEN
	M_isDone := TRUE;
ELSE 
	M_isDone := FALSE;
END_IF
END_METHOD

METHOD PUBLIC M_Tuerablaufstarten : BOOL
VAR_INPUT
	m_Stockwerk : INT;
END_VAR
IF m_Stockwerk >= 1 AND m_Stockwerk <= 6 THEN
	TuerzyklusStarten := TRUE;
	Stockwerk := m_Stockwerk;
	M_Tuerablaufstarten := TRUE;
ELSE
	M_Tuerablaufstarten := FALSE;
END_IF
END_METHOD

END_FUNCTION_BLOCK

// ---- 0_App/Lib/FB_Achse.TcPOU
FUNCTION_BLOCK FB_Achse
VAR_INPUT
	Simulation : BOOL; //Bei True wird über S_Zielposition die Zielpostion manuell übergeben
	S_Zielposition : LREAL; //Zielpostion zum Testen des Bausteins
	

END_VAR
VAR_OUTPUT
END_VAR
VAR
	FehlercodePower : UDINT;
	FehlercodeMove : UDINT;
	FehlercodeRef: UDINT;
	State :ENUM_Achse;
	Zielposition : LREAL;
	Start : BOOL;
	AktuellePosition : LREAL;
	Referenzieren : BOOL;
	MoveAbsExecute : BOOL;
	HomeExecute : BOOL;
	ResetExecute : BOOL;
	PowerExecute : BOOL;
	Error	: BOOL;
	Done	: BOOL;
	Busy 	: BOOL;
	AchseReset :BOOL;
	fbPower    : MC_Power;
    fbHome     : MC_Home;
    fbMoveAbs  : MC_MoveAbsolute;
    fbStop     : MC_Stop;
    fbReset    : MC_Reset;
	fbJog   : MC_Jog;
	fbReadPos : MC_ReadActualPosition;
	AchseReferenzieren : BOOL;
	s_Zielstock : INT;

END_VAR
VAR_IN_OUT
	Achse : AXIS_REF;
END_VAR

fbPower(
		Axis:= Achse, 
		Enable:= PowerExecute, 
		Enable_Positive:= TRUE, 
		Enable_Negative:= TRUE,  
		ErrorID => FehlercodePower);
fbReadPos(
    Axis    := Achse,
    Enable  := TRUE,
    Position => Divers.AktuellePosmm  // ← schreibt jeden Zyklus die Position in mm
);
		
fbJog(
    Axis         := Achse,
    JogForward   := Visu_Manuellmodus.JogAuf AND Divers.ManuellmodusAktiv AND fbPower.Status,
    JogBackwards := Visu_Manuellmodus.JogAb  AND Divers.ManuellmodusAktiv AND fbPower.Status,
    Velocity     := 100.0   // mm/s – anpassen nach Bedarf
);
IF Simulation THEN
		Zielposition := S_Zielposition;
	END_IF
	
CASE State OF
		ENUM_Achse.Warten: // Achse nicht eingeschalten 
		Error := FALSE;
		Divers.AchseSicher := TRUE;
		IF Start AND NOT fbPower.Status THEN
			Divers.AchseSicher := FALSE;
			Start := FALSE;
			Done := FALSE;
			Busy := TRUE;
			ResetExecute := TRUE;
			State := ENUM_Achse.PowerOn;
		END_IF
		IF Start AND fbPower.Status THEN
			Divers.AchseSicher := FALSE;
			Start := FALSE;
			Done := FALSE;
			Busy := TRUE;
			MoveAbsExecute := TRUE;
			State := ENUM_Achse.Positionieren;
		END_IF
		IF AchseReferenzieren AND fbPower.Status THEN //Falls Fahrsystem Referenzierung durchführen will
			AchseReferenzieren := FALSE;
			Done := FALSE;
			Busy := TRUE;
			HomeExecute := TRUE;
			State := ENUM_Achse.Referenzieren;
		END_IF
		IF AchseReferenzieren AND NOT fbPower.Status THEN //Falls Fahrsystem Referenzierung durchführen will
			Divers.AchseSicher := FALSE;
			AchseReferenzieren := FALSE;
			Done := FALSE;
			Busy := TRUE;
			ResetExecute := TRUE;
			State := ENUM_Achse.PowerOn;
		END_IF
		
	ENUM_Achse.PowerOn: // Achse einschalten

		PowerExecute := TRUE;
		
			 
		IF fbPower.Status THEN
			HomeExecute := TRUE;
			State := ENUM_Achse.Referenzieren;
		END_IF
		IF fbPower.Error THEN
			Busy := FALSE;
			Error := TRUE; 
			HomeExecute := FALSE;
			State := ENUM_Achse.Error;
		END_IF
		
	ENUM_Achse.Referenzieren:
	
			fbHome(
			Axis:= Achse , 
			Execute:= HomeExecute , 
			Position:= 0.0, 
			HomingMode:= MC_DefaultHoming, 
			bCalibrationCam := IO_L1.Control_LiftAxisReference,
			ErrorID => FehlercodeRef
			 );
			
		IF fbHome.Busy THEN
			HomeExecute := FALSE;
		END_IF

	
		IF fbHome.Done THEN
			Done := TRUE;
			Busy := FALSE;
			State := ENUM_Achse.Warten;
		END_IF
		IF fbHome.Error THEN
			Error := TRUE;
			State := ENUM_Achse.Error;
		END_IF
		
	ENUM_Achse.Positionieren:
		fbMoveAbs(
			Axis:= Achse, 
			Execute:= MoveAbsExecute, 
			Position:= Zielposition, 
			Velocity:= 400.0 , //Kein plan wie gross der Wert sein sollte
			ErrorID => FehlercodeMove
			 );
			 
		MoveAbsExecute := FALSE;
		IF fbMoveAbs.Done THEN
			Divers.AktuellesStockwerk := s_Zielstock;
			Done := TRUE;
			Busy := FALSE;
			State := ENUM_Achse.Warten;
		END_IF
		IF fbMoveAbs.Error THEN
			Done := FALSE;
			Busy := FALSE;
			Error := TRUE;
			State := ENUM_Achse.Error;
		END_IF
			
	ENUM_Achse.Error:  //Bedinung einfügen, um aus Error zu kommen
		Error := TRUE;
		IF IO_L1.Control_Reset THEN
			AchseReset := TRUE; 
			fbReset(
				Axis:= Achse , 
				Execute:= AchseReset, 
				Done=> , 
				Busy=> , 
				Error=> Error, 
				ErrorID=> );
				
			IF fbReset.Done THEN
				AchseReset := FALSE;
				State := ENUM_Achse.Warten;
			END_IF
		END_IF
END_CASE

METHOD PUBLIC M_AufstartenAbgeschlossen : BOOL
VAR_INPUT
END_VAR
END_METHOD

METHOD PRIVATE M_getDirection : BOOL
VAR_INPUT
	md_Zielposition : LREAL;
END_VAR
IF md_Zielposition > AktuellePosition THEN
	M_getDirection := TRUE;
END_IF
IF md_Zielposition < AktuellePosition THEN
	M_getDirection := FALSE;
END_IF
END_METHOD

METHOD PUBLIC M_getPosition : LREAL
VAR_INPUT
END_VAR
M_getPosition := AktuellePosition;
END_METHOD

METHOD PUBLIC M_hasError : BOOL
VAR_INPUT
END_VAR
IF Error THEN
	M_hasError := TRUE;
ELSE
	M_hasError := FALSE;
END_IF
END_METHOD

METHOD M_isBusy : BOOL
VAR_INPUT
END_VAR
IF Busy THEN
	M_isBusy := TRUE;
ELSE
	M_isBusy := FALSE;
END_IF
END_METHOD

METHOD M_isDone : BOOL
VAR_INPUT
END_VAR
IF Done THEN
	M_isDone := TRUE;
ELSE
	M_isDone := FALSE;
END_IF
END_METHOD

METHOD PUBLIC M_Movetoposition : BOOL
VAR_INPUT
	ZielStock : INT;
END_VAR
IF NOT Busy AND NOT Error THEN
	Zielposition := FC_GetFloorPosition(ZielStock);
	s_Zielstock := ZielStock;
	Start := TRUE;
	M_Movetoposition := TRUE; //Rückgabewert
ELSE
	M_Movetoposition := FALSE;
END_IF
END_METHOD

METHOD PUBLIC M_Referenzieren : BOOL
VAR_INPUT
END_VAR
IF (Done) THEN
	AchseReferenzieren := TRUE;
	M_Referenzieren := TRUE;
ELSE
	M_Referenzieren := FALSE;
END_IF
END_METHOD

END_FUNCTION_BLOCK

// ---- 0_App/Lib/FC_GetFloorPosition.TcPOU
FUNCTION FC_GetFloorPosition : LREAL
VAR_INPUT
	Stockwerk : INT;
END_VAR
VAR
	Stockwerkpositionen : ARRAY[1..6] OF LREAL := [60.0, 300.0, 540.0, 770.0, 1020.0, 1250.0]; //fiktionale Werte
END_VAR
// Dieser Funktion kann man das Stockwerk übergeben und es wird die Achsposition zurückgegeben
// Also z.B Stock 5 --> 1250mm 
// So können wir die Werte ermitteln mit testen und hier eintragen und nicht irgendwo im programm versteckt

IF (Stockwerk >= 1) AND (Stockwerk <= 6) THEN
    FC_GetFloorPosition := Stockwerkpositionen[Stockwerk];
ELSE
    FC_GetFloorPosition := 0.0; // oder irgend ein Fehler
END_IF

END_FUNCTION

// ---- 0_App/Lib/FB_Blinker.TcPOU
FUNCTION_BLOCK FB_Blinker
VAR_INPUT
    bEnable : BOOL := TRUE;
    tOn     : TIME := T#500MS;
    tOff    : TIME := T#500MS;
END_VAR

VAR_OUTPUT
    bOut : BOOL;
END_VAR

VAR
    tonOn  : TON;
    tonOff : TON;
END_VAR

IF NOT bEnable THEN
    bOut := FALSE;
    tonOn(IN := FALSE);
    tonOff(IN := FALSE);
ELSE
    IF bOut THEN
        tonOn(IN := TRUE, PT := tOn);
        tonOff(IN := FALSE);

        IF tonOn.Q THEN
            bOut := FALSE;
            tonOn(IN := FALSE);
        END_IF
    ELSE
        tonOff(IN := TRUE, PT := tOff);
        tonOn(IN := FALSE);

        IF tonOff.Q THEN
            bOut := TRUE;
            tonOff(IN := FALSE);
        END_IF
    END_IF
END_IF

END_FUNCTION_BLOCK

// ---- 0_App/Lib/FB_Manuell.TcPOU
FUNCTION_BLOCK FB_Manuell
VAR_INPUT
	
	
	
END_VAR
VAR_OUTPUT

	
END_VAR
VAR
i : INT;
END_VAR

FOR i := 1 TO 6 DO

    IF i = Visu_Manuellmodus.Zielstock THEN
        Visu_Manuellmodus.adwFloorBtnColor[i] := 16#FFFF8000;  // Orange, opak
    ELSE
       Visu_Manuellmodus.adwFloorBtnColor[i] := 16#FFFFFFFF;  // Weiss, opak
    END_IF

    // Tür-Buttons bleiben unverändert
    IF Visu_Manuellmodus.bTuerAuf[i] THEN
        Visu_Manuellmodus.adwTuerAufColor[i] := 16#FF0000FF;
    ELSE
        Visu_Manuellmodus.adwTuerAufColor[i] := 16#FF808080;
    END_IF
    IF Visu_Manuellmodus.bTuerZu[i] THEN
        Visu_Manuellmodus.adwTuerZuColor[i] := 16#FF0000FF;
    ELSE
        Visu_Manuellmodus.adwTuerZuColor[i] := 16#FF808080;
    END_IF

END_FOR

END_FUNCTION_BLOCK

// ---- 0_App/Lib/FB_Taskmanager_1.TcPOU
FUNCTION_BLOCK FB_Taskmanager_1
VAR_INPUT
	 fbFahrlogik      : ITF_Fahrlogik;
END_VAR
VAR_IN_OUT
	fbFahrleitsystem : FB_Fahrleitsystem;
	
END_VAR
VAR_OUTPUT
END_VAR
VAR
	
   
	nextFree	:	INT;
	Auftraege : ARRAY[1..10] OF ST_Fahrauftrag; //bin was am probieren
	
	State : INT;
	StartLogik:	BOOL;
	NextTask	:	ST_Fahrauftrag;
END_VAR

IF Auftraege[1].istAktiv AND NOT fbFahrleitsystem.M_isBusy() THEN
	StartLogik := TRUE;
END_IF

Case State Of
	
00: //Warten
IF StartLogik AND IO_L1.Control_Automatic THEN
	StartLogik := FALSE;
	State := 10;
END_IF

//-------------------------------------------------------------------------------------------------

10: //Nächste Task von der Fahrlogik geben lassen
NextTask := fbFahrlogik.M_getNextTask(
Divers.AktuellesStockwerk, Auftraege);

IF NextTask.Auftragsnummer > 0 THEN
	State := 20;
ELSE
	State := 0;
END_IF

//-------------------------------------------------------------------------------------------------

20://Task dem Fahrleitsystem übergeben
IF NOT fbFahrleitsystem.M_isBusy() THEN 
		IF fbFahrleitsystem.M_AcceptTask(NextTask) THEN
            State := 30; 
        END_IF
END_IF

//-------------------------------------------------------------------------------------------------
30:

        IF fbFahrleitsystem.M_isDone() THEN
            State := 40;
        END_IF

//----------------------------------------------------------------------------------------------------

40: //Alles zurücksetzten auftrag löschen und wieder in State 1 gehen
	IF M_deleteFinishedTask(TaskToDelete :=  NextTask) THEN
		State:=00;
	END_IF

END_CASE

METHOD M_deleteFinishedTask : BOOL
VAR_INPUT
	TaskToDelete : ST_Fahrauftrag;
	
END_VAR
VAR
	i:DINT;
	j:DINT;
	IndextoDelete : DINT;
END_VAR
FOR j:=1 TO UPPER_BOUND(Auftraege, 1) DO
	IF TaskToDelete.Auftragsnummer	= Auftraege[j].Auftragsnummer AND Auftraege[j].istAktiv THEN  
		IndextoDelete := j;
		EXIT;
	END_IF
END_FOR

IF IndextoDelete > 0 THEN
	FOR i := IndextoDelete TO (UPPER_BOUND(Auftraege,1)-1) DO
		Auftraege[i] := Auftraege[i+1];
	END_FOR

	Auftraege[UPPER_BOUND(Auftraege,1)].istAktiv	:= FALSE;
	Auftraege[UPPER_BOUND(Auftraege,1)].Auftragsnummer := 0;
	Auftraege[UPPER_BOUND(Auftraege,1)].Startstockwerk := 0;
	Auftraege[UPPER_BOUND(Auftraege,1)].Zielstockwerk	:= 0;

	M_deleteFinishedTask := TRUE;
ELSE
	M_deleteFinishedTask := FALSE;
END_IF
END_METHOD

METHOD PUBLIC M_newTask : BOOL
VAR_INPUT
	Start	:	INT;
	Ziel	:	INT;
END_VAR
VAR
	
	Accept : BOOL; // nur test
	i:INT;
END_VAR

FOR i:=1 TO 10 DO
	IF NOT Auftraege[i].istAktiv THEN
		Auftraege[i].Startstockwerk := Start;
		Auftraege[i].Zielstockwerk := Ziel;
		
		Divers.NextfreeOrderID := Divers.NextfreeOrderID + 1;
		Auftraege[i].Auftragsnummer := Divers.NextfreeOrderID;
		
		Auftraege[i].istAktiv := TRUE;
		StartLogik := TRUE;
		M_newTask := TRUE;
		
		EXIT;
	END_IF
END_FOR
END_METHOD

METHOD PUBLIC M_TaskDone : BOOL
VAR_INPUT
	
END_VAR
VAR_IN_OUT
	
END_VAR
END_METHOD

END_FUNCTION_BLOCK

// ---- 0_App/Lib/Diverses/FB_Logik_FIFO.TcPOU
FUNCTION_BLOCK FB_Logik_FIFO IMPLEMENTS ITF_Fahrlogik
VAR_INPUT
END_VAR
VAR_OUTPUT
END_VAR
VAR
END_VAR

{warning 'Methodenimplementierung hinzufügen'}
METHOD M_getNextTask : ST_Fahrauftrag
VAR_INPUT
	LiftStockwerkAktuell	: INT;
END_VAR
VAR_IN_OUT
	Auftraege	: ARRAY [1..10] OF ST_Fahrauftrag;
END_VAR


IF Auftraege[1].istAktiv THEN
    M_getNextTask := Auftraege[1];
ELSE
    // Wenn nichts da ist, geben wir einen leeren Struct zurück
    M_getNextTask.Auftragsnummer := 0; 
END_IF
END_METHOD

END_FUNCTION_BLOCK

// ---- 0_App/Lib/Diverses/FB_Logik_ShortestDistance.TcPOU
FUNCTION_BLOCK FB_Logik_ShortestDistance IMPLEMENTS ITF_Fahrlogik
VAR_INPUT
END_VAR
VAR_OUTPUT
END_VAR
VAR
END_VAR

{warning 'Methodenimplementierung hinzufügen'}
METHOD M_getNextTask : ST_Fahrauftrag
VAR_INPUT
	LiftStockwerkAktuell	: INT;
END_VAR
VAR_IN_OUT
	(* Die Liste zum Durchsuchen*)
	Auftraege	: ARRAY [1..10] OF ST_Fahrauftrag;
END_VAR
VAR
	i : DINT;
    BestIndex : DINT := 0;
    shortestDistance  : INT := 100; // Startwert extrem hoch setzen
    Distance     : INT;
    Leer       : ST_Fahrauftrag;
END_VAR

FOR i := 1 TO UPPER_BOUND(Auftraege, 1) DO
	
IF Auftraege[i].istAktiv THEN
	Distance := ABS(Auftraege[i].Startstockwerk - Divers.AktuellesStockwerk);
	
	IF Distance < shortestDistance THEN
		shortestDistance := Distance;
		BestIndex := i;
	END_IF
END_IF
END_FOR

IF BestIndex > 0 THEN
	M_getNextTask := Auftraege[BestIndex];
ELSE
	M_getNextTask := Leer;
END_IF
END_METHOD

END_FUNCTION_BLOCK

// ---- 0_App/Lib/FB_Panel.TcPOU
FUNCTION_BLOCK FB_Panel
VAR_INPUT
Panel_1_Btn : ARRAY[1..6] OF BOOL; // Panel Level 1 - Buttons
Panel_2_Btn : ARRAY[1..6] OF BOOL; // Panel Level 2 - Buttons
Panel_3_Btn : ARRAY[1..6] OF BOOL; // Panel Level 3 - Buttons
Panel_4_Btn : ARRAY[1..6] OF BOOL; // Panel Level 4 - Buttons
Panel_5_Btn : ARRAY[1..6] OF BOOL; // Panel Level 5 - Buttons
Panel_6_Btn : ARRAY[1..6] OF BOOL; // Panel Level 6 - Buttons


END_VAR
VAR_OUTPUT
	//LEDS
	Panel_1_BtnLED : ARRAY[1..6] OF BOOL;
	Panel_2_BtnLED : ARRAY[1..6] OF BOOL;
	Panel_3_BtnLED : ARRAY[1..6] OF BOOL;
	Panel_4_BtnLED : ARRAY[1..6] OF BOOL;
	Panel_5_BtnLED : ARRAY[1..6] OF BOOL;
	Panel_6_BtnLED : ARRAY[1..6] OF BOOL;
	
	Panel_1_Led_Up  : BOOL;
	Panel_1_Led_Down: BOOL;
	Panel_2_Led_Up  : BOOL;
	Panel_2_Led_Down: BOOL;
	Panel_3_Led_Up  : BOOL;
	Panel_3_Led_Down: BOOL;
	Panel_4_Led_Up  : BOOL;
	Panel_4_Led_Down: BOOL;
	Panel_5_Led_Up  : BOOL;
	Panel_5_Led_Down: BOOL;
	Panel_6_Led_Up  : BOOL;
	Panel_6_Led_Down: BOOL;
	
	//7-Segment-Anzeige
	Panel_1_BCD_Bit : ARRAY[0..3] OF BOOL;
	Panel_2_BCD_Bit : ARRAY[0..3] OF BOOL;
	Panel_3_BCD_Bit : ARRAY[0..3] OF BOOL;
	Panel_4_BCD_Bit : ARRAY[0..3] OF BOOL;
	Panel_5_BCD_Bit : ARRAY[0..3] OF BOOL;
	Panel_6_BCD_Bit : ARRAY[0..3] OF BOOL;
END_VAR
VAR_IN_OUT
	fbTaskManager : FB_Taskmanager_1;
	
END_VAR
VAR
Panel_Btn : ARRAY[1..6] OF ARRAY [1..6] OF BOOL;
TrigBtn : ARRAY[1..6] OF ARRAY [1..6] OF R_TRIG;

meinStockwerk	:	INT;
meinZiel		:	INT;
AuftragAngenommen : BOOL;

//LED
Panel_LEDs	:	ARRAY[1..6] OF ARRAY[1..6] OF BOOL;
Panel_LED_UP:	ARRAY[1..6] OF BOOL;
Panel_LED_Down:	ARRAY[1..6] OF BOOL;

//7-Segment
Panel_BCD	:	ARRAY[1..6] OF ARRAY[0..3] OF BOOL;

//LED's löschen
PanelLED_loeschen : INT;
LED_loeschen : BOOL;

END_VAR

//Stockwerkbuttons
Panel_Btn[1] := Panel_1_Btn;
Panel_Btn[2] := Panel_2_Btn;
Panel_Btn[3] := Panel_3_Btn;
Panel_Btn[4] := Panel_4_Btn;
Panel_Btn[5] := Panel_5_Btn;
Panel_Btn[6] := Panel_6_Btn;


FOR meinStockwerk := 1 TO 6 DO
	FOR meinZiel := 1 TO 6 DO
			TrigBtn[meinStockwerk][meinZiel](CLK := Panel_Btn[meinStockwerk][meinZiel]);
        	IF TrigBtn[meinStockwerk][meinZiel].Q THEN
			 	AuftragAngenommen := fbTaskManager.M_newTask(Start := meinStockwerk, Ziel := meinZiel);
				
				IF AuftragAngenommen THEN
                Panel_LEDs[meinStockwerk][meinZiel] := TRUE;
					IF meinStockwerk < meinZiel THEN
						Panel_LED_UP[meinStockwerk] := TRUE;
					END_IF
					IF meinStockwerk > meinZiel THEN
						Panel_LED_Down[meinStockwerk] := TRUE;
					END_IF
				
				//BCD
				Panel_BCD[meinStockwerk][0] := meinZiel.0; // Bit 0 (Wertigkeit 1)
    			Panel_BCD[meinStockwerk][1] := meinZiel.1; // Bit 1 (Wertigkeit 2)
    			Panel_BCD[meinStockwerk][2] := meinZiel.2; // Bit 2 (Wertigkeit 4)
    			Panel_BCD[meinStockwerk][3] := meinZiel.3; // Bit 3 (Wertigkeit 8)
				
           		 ELSE
                // Fehlermanagement
            END_IF
        END_IF
	END_FOR
END_FOR
//LED's zurücksetzen
IF LED_loeschen THEN
	Panel_LEDs[Divers.AktuellesStockwerk][PanelLED_loeschen] := FALSE;
	Panel_LED_UP[Divers.AktuellesStockwerk] := FALSE;
	panel_LED_DOWN[Divers.AktuellesStockwerk] := FALSE;
	Panel_BCD[Divers.AktuellesStockwerk][0] := 0;
	Panel_BCD[Divers.AktuellesStockwerk][1] := 0;
	Panel_BCD[Divers.AktuellesStockwerk][2] := 0;
	Panel_BCD[Divers.AktuellesStockwerk][3] := 0;
	LED_loeschen := FALSE;
END_IF

//Stockwerk LEDs
Panel_1_BtnLED := Panel_LEDs[1];
Panel_2_BtnLED := Panel_LEDs[2];
Panel_3_BtnLED := Panel_LEDs[3];
Panel_4_BtnLED := Panel_LEDs[4];
Panel_5_BtnLED := Panel_LEDs[5];
Panel_6_BtnLED := Panel_LEDs[6];

// Hoch LEDs
Panel_1_Led_Up := Panel_LED_UP[1];
Panel_2_Led_Up := Panel_LED_UP[2];
Panel_3_Led_Up := Panel_LED_UP[3];
Panel_4_Led_Up := Panel_LED_UP[4];
Panel_5_Led_Up := Panel_LED_UP[5];
Panel_6_Led_Up := Panel_LED_UP[6];

// Runter LEDs
Panel_1_Led_Down := Panel_LED_Down[1];
Panel_2_Led_Down := Panel_LED_Down[2];
Panel_3_Led_Down := Panel_LED_Down[3];
Panel_4_Led_Down := Panel_LED_Down[4];
Panel_5_Led_Down := Panel_LED_Down[5];
Panel_6_Led_Down := Panel_LED_Down[6];

//BCD
Panel_1_BCD_Bit := Panel_BCD[1];
Panel_2_BCD_Bit := Panel_BCD[2];
Panel_3_BCD_Bit := Panel_BCD[3];
Panel_4_BCD_Bit := Panel_BCD[4];
Panel_5_BCD_Bit := Panel_BCD[5];
Panel_6_BCD_Bit := Panel_BCD[6];

METHOD PUBLIC M_TurnofLED : BOOL
VAR_INPUT
	Stockwerk_LED_Loeschen : INT;
END_VAR
PanelLED_loeschen := Stockwerk_LED_Loeschen; //PanelLED_loeschen = Knopf 1-6, von dem LEDs gelöscht werden sollen
LED_loeschen := TRUE;
M_TurnofLED := TRUE;
END_METHOD

END_FUNCTION_BLOCK

// ---- 7_Visu/Common/Control.TcVIS
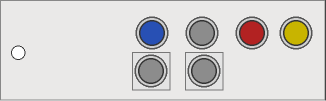
VISUALIZATION Control  // 326x101
VAR_IN_OUT
	LED_Blue : BOOL;
	LED_Red : BOOL;
	LED_White : BOOL;
	LED_Yellow : BOOL;
	Start : BOOL;
	Reset : BOOL;
	State : INT;
END_VAR
    Rectangle (0,0 326x100)
    Lamp1 (276,14 40x38), variable: LED_Yellow, style: Lamp-Lamp1-Yellow
    PushSwitch (182,52 44x38), variable: Start, behaviour: TAP, style: Switch-PushSwitch-Gray
    RadioButton (9,4 122x97), variable: State
        Areas[0]: Text=Off
        Areas[1]: Text=Manual
        Areas[2]: Text=Automatic
    Lamp1 (132,14 40x38), variable: LED_Blue, style: Lamp-Lamp1-Blue
    Lamp1 (232,14 40x38), variable: LED_Red, style: Lamp-Lamp1-Red
    Lamp1 (182,14 40x38), variable: LED_White, style: Lamp-Lamp1-Gray
    PushSwitch (129,52 44x38), variable: Reset, behaviour: TAP, style: Switch-PushSwitch-Gray
END_VISUALIZATION

// ---- 7_Visu/Common/Floor.TcVIS
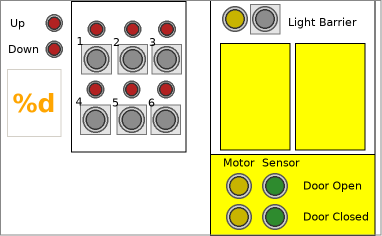
VISUALIZATION Floor  // 382x236
VAR_IN_OUT
	Color 			: DWORD;
	LED_Up	 		: BOOL;
	LED_Down		: BOOL;
	FloorNumber 	: INT;
	BtnLed	 		: ARRAY[1..6] OF BOOL;;
	Btn				: ARRAY[1..6] OF BOOL;
	LB	 			: BOOL;
	LED_DoorOpen 	: BOOL;
	LED_DoorClosed	: BOOL;
	PositionDoor	: REAL;
	M_Open 			: BOOL;
	M_Close			: BOOL;
END_VAR
    Frame (0,0 186x152)
        shows FloorControl(LED_Up := LED_Up, LED_Down := LED_Down, FloorNumber := FloorNumber, BtnLed := BtnLed, Btn := Btn)
    Rectangle (210,0 165x236)
    Rectangle (210,154 165x82), colour variable: Color
    Rectangle (295,43 70x107), colour variable: Color
        p3560616238: (40/100.0*PositionDoor)
    Rectangle (220,43 70x107), colour variable: Color
        p3560616238: -(40/100.0*PositionDoor)
    Lamp1 (260,171 30x30), variable: LED_DoorOpen, style: Lamp-Lamp1-Green
    Lamp1 (260,202 30x30), variable: LED_DoorClosed, style: Lamp-Lamp1-Green
    Label (300,171 82x30), "Door Open"
    Label (300,202 82x30), "Door Closed"
    Label (285,11 82x23), "Light Barrier"
    Lamp1 (220,4 30x30), variable: LB, style: Lamp-Lamp1-Yellow
    PushSwitch (250,4 30x30), variable: LB, behaviour: TAP, style: Switch-PushSwitch-Gray
    Lamp1 (224,202 30x30), variable: M_Close, style: Lamp-Lamp1-Yellow
    Lamp1 (224,171 30x30), variable: M_Open, style: Lamp-Lamp1-Yellow
    Label (220,148 41x30), "Motor"
    Label (259,148 41x30), "Sensor"
END_VISUALIZATION

// ---- 7_Visu/Common/FloorControl.TcVIS
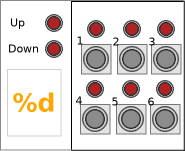
VISUALIZATION FloorControl  // 185x151
VAR_IN_OUT
	LED_Up	 		: BOOL;
	LED_Down		: BOOL;
	FloorNumber 	: INT;
	BtnLed	 		: ARRAY[1..6] OF BOOL;;
	Btn				: ARRAY[1..6] OF BOOL;
END_VAR
    RoundedRectangle (71,1 114x150)
    PushSwitch (81,44 30x30), variable: Btn[1], behaviour: TAP, style: Switch-PushSwitch-Gray
    Lamp1 (86,19 20x20), variable: BtnLed[1], style: Lamp-Lamp1-Red
    PushSwitch (117,44 30x30), variable: Btn[2], behaviour: TAP, style: Switch-PushSwitch-Gray
    Lamp1 (122,19 20x20), variable: BtnLed[2], style: Lamp-Lamp1-Red
    PushSwitch (151,44 30x30), variable: Btn[3], behaviour: TAP, style: Switch-PushSwitch-Gray
    Lamp1 (156,19 20x20), variable: BtnLed[3], style: Lamp-Lamp1-Red
    Lamp1 (44,13 20x20), variable: LED_Up, style: Lamp-Lamp1-Red
    Lamp1 (44,39 20x20), variable: LED_Down, style: Lamp-Lamp1-Red
    Label (70,31 20x20), "1"
    Label (106,32 20x20), "2"
    Label (142,32 20x20), "3"
    PushSwitch (80,104 30x30), variable: Btn[4], behaviour: TAP, style: Switch-PushSwitch-Gray
    Lamp1 (85,79 20x20), variable: BtnLed[4], style: Lamp-Lamp1-Red
    PushSwitch (116,104 30x30), variable: Btn[5], behaviour: TAP, style: Switch-PushSwitch-Gray
    Lamp1 (121,79 20x20), variable: BtnLed[5], style: Lamp-Lamp1-Red
    PushSwitch (150,104 30x30), variable: Btn[6], behaviour: TAP, style: Switch-PushSwitch-Gray
    Lamp1 (155,79 20x20), variable: BtnLed[6], style: Lamp-Lamp1-Red
    Label (69,91 20x20), "4"
    Label (105,92 20x20), "5"
    Label (141,92 20x20), "6"
    Label (7,13 36x20), "Up"
    Label (5,39 38x20), "Down"
    Textfield (7,69 54x67), "%d", text variable: FloorNumber
END_VISUALIZATION

// ---- 7_Visu/Common/Lift.TcVIS
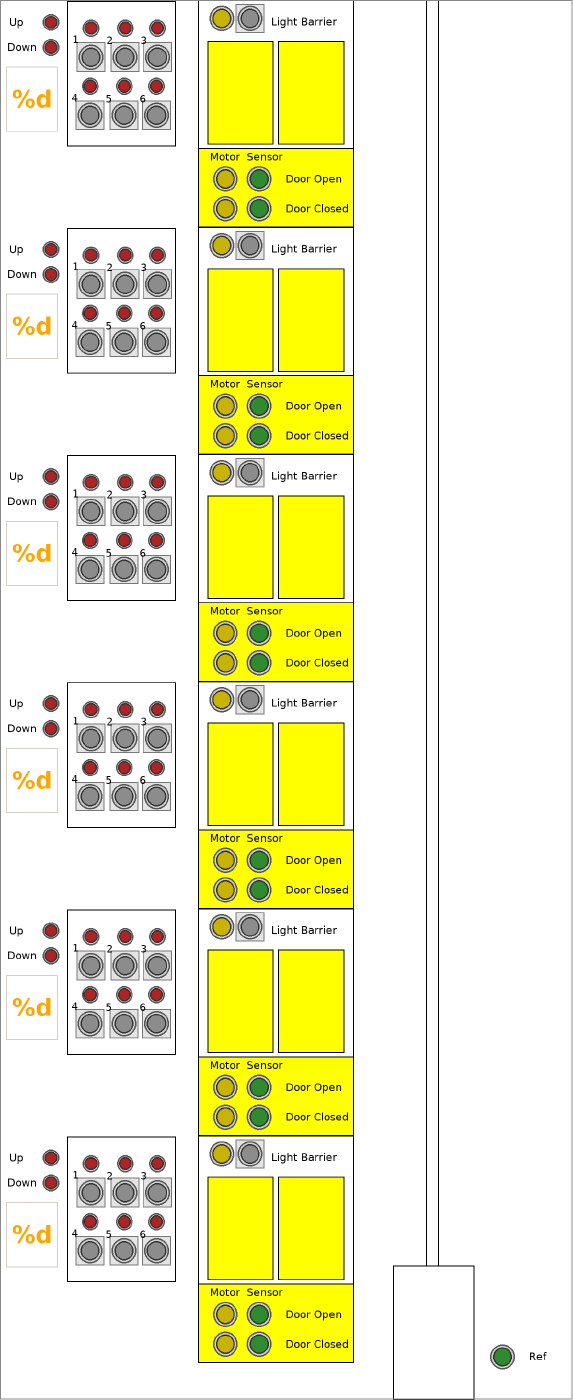
VISUALIZATION Lift  // 598x1461
VAR_IN_OUT
	Position : REAL;
	RefSensor : BOOL;
	Color : DWORD;
	Door_1_Position	: REAL;
	Door_1_M_Open	: BOOL;
	Door_1_M_Close	: BOOL;
	Door_2_Position	: REAL;
	
	Door_2_M_Open	: BOOL;
	Door_2_M_Close	: BOOL;
	Door_3_Position	: REAL;
	
	Door_3_M_Open	: BOOL;
	Door_3_M_Close	: BOOL;
	Door_4_Position	: REAL;
	
	Door_4_M_Open	: BOOL;
	Door_4_M_Close	: BOOL;
	Door_5_Position	: REAL;
	
	Door_5_M_Open	: BOOL;
	Door_5_M_Close	: BOOL;
	Door_6_Position	: REAL;
	
	Door_6_M_Open	: BOOL;
	Door_6_M_Close	: BOOL;
	LED_Up_1 		: BOOL;
	LED_Down_1 		: BOOL;
	FloorNumber_1 	: INT;
	BtnLed_1 		: ARRAY[1..6] OF BOOL;;
	Btn_1			: ARRAY[1..6] OF BOOL;
	LB_1 			: BOOL;
	LED_DoorOpen_1 	: BOOL;
	LED_DoorClosed_1: BOOL;

	LED_Up_2 		: BOOL;
	LED_Down_2 		: BOOL;
	FloorNumber_2 	: INT;
	BtnLed_2 		: ARRAY[1..6] OF BOOL;;
	Btn_2			: ARRAY[1..6] OF BOOL;
	LB_2 			: BOOL;
	LED_DoorOpen_2 	: BOOL;
	LED_DoorClosed_2: BOOL;


	LED_Up_3 		: BOOL;
	LED_Down_3 		: BOOL;
	FloorNumber_3 	: INT;
	BtnLed_3 		: ARRAY[1..6] OF BOOL;;
	Btn_3			: ARRAY[1..6] OF BOOL;
	LB_3 			: BOOL;
	LED_DoorOpen_3 	: BOOL;
	LED_DoorClosed_3: BOOL;

	LED_Up_4 		: BOOL;
	LED_Down_4 		: BOOL;
	FloorNumber_4 	: INT;
	BtnLed_4 		: ARRAY[1..6] OF BOOL;;
	Btn_4			: ARRAY[1..6] OF BOOL;
	LB_4 			: BOOL;
	LED_DoorOpen_4 	: BOOL;
	LED_DoorClosed_4: BOOL;

	LED_Up_5 		: BOOL;
	LED_Down_5 		: BOOL;
	FloorNumber_5 	: INT;
	BtnLed_5 		: ARRAY[1..6] OF BOOL;;
	Btn_5			: ARRAY[1..6] OF BOOL;
	LB_5 			: BOOL;
	LED_DoorOpen_5 	: BOOL;
	LED_DoorClosed_5: BOOL;

	LED_Up_6 		: BOOL;
	LED_Down_6 		: BOOL;
	FloorNumber_6 	: INT;
	BtnLed_6 		: ARRAY[1..6] OF BOOL;;
	Btn_6			: ARRAY[1..6] OF BOOL;
	LB_6 			: BOOL;
	LED_DoorOpen_6 	: BOOL;
	LED_DoorClosed_6: BOOL;

END_VAR
    Frame (410,0 188x1461)
        shows Lift_Axis(Position := Visu_L1.Position_LIFT, RefSensor := RefSensor)
    Frame (0,0 376x1422)
        shows Lift_Floors(Color := Color, Door_1_Position := Door_1_Position, Door_1_M_Open := Door_1_M_Open, Door_1_M_Close := Door_1_M_Close, Door_2_Position := Door_2_Position, Door_2_M_Open := Door_2_M_Open, Door_2_M_Close := Door_2_M_Close, Door_3_Position := Door_3_Position, Door_3_M_Open := Door_3_M_Open, Door_3_M_Close := Door_3_M_Close, Door_4_Position := Door_4_Position, Door_4_M_Open := Door_4_M_Open, Door_4_M_Close := Door_4_M_Close, Door_5_Position := Door_5_Position, Door_5_M_Open := Door_5_M_Open, Door_5_M_Close := Door_5_M_Close, Door_6_Position := Door_6_Position, Door_6_M_Open := Door_6_M_Open, Door_6_M_Close := Door_6_M_Close, LED_Up_1 := LED_Up_1, LED_Down_1 := LED_Down_1, FloorNumber_1 := FloorNumber_1, BtnLed_1 := BtnLed_1, Btn_1 := Btn_1, LB_1 := LB_1, LED_DoorOpen_1 := LED_DoorOpen_1, LED_DoorClosed_1 := LED_DoorClosed_1, LED_Up_2 := LED_Up_2, LED_Down_2 := LED_Down_2, FloorNumber_2 := FloorNumber_2, BtnLed_2 := BtnLed_2, Btn_2 := Btn_2, LB_2 := LB_2, LED_DoorOpen_2 := LED_DoorOpen_2, LED_DoorClosed_2 := LED_DoorClosed_2, LED_Up_3 := LED_Up_3, LED_Down_3 := LED_Down_3, FloorNumber_3 := FloorNumber_3, BtnLed_3 := BtnLed_3, Btn_3 := Btn_3, LB_3 := LB_3, LED_DoorOpen_3 := LED_DoorOpen_3, LED_DoorClosed_3 := LED_DoorClosed_3, LED_Up_4 := LED_Up_4, LED_Down_4 := LED_Down_4, FloorNumber_4 := FloorNumber_4, BtnLed_4 := BtnLed_4, Btn_4 := Btn_4, LB_4 := LB_4, LED_DoorOpen_4 := LED_DoorOpen_4, LED_DoorClosed_4 := LED_DoorClosed_4, LED_Up_5 := LED_Up_5, LED_Down_5 := LED_Down_5, FloorNumber_5 := FloorNumber_5, BtnLed_5 := BtnLed_5, Btn_5 := Btn_5, LB_5 := LB_5, LED_DoorOpen_5 := LED_DoorOpen_5, LED_DoorClosed_5 := LED_DoorClosed_5, LED_Up_6 := LED_Up_6, LED_Down_6 := LED_Down_6, FloorNumber_6 := FloorNumber_6, BtnLed_6 := BtnLed_6, Btn_6 := Btn_6, LB_6 := LB_6, LED_DoorOpen_6 := LED_DoorOpen_6, LED_DoorClosed_6 := LED_DoorClosed_6)
END_VISUALIZATION

// ---- 7_Visu/Common/Lift_Axis.TcVIS
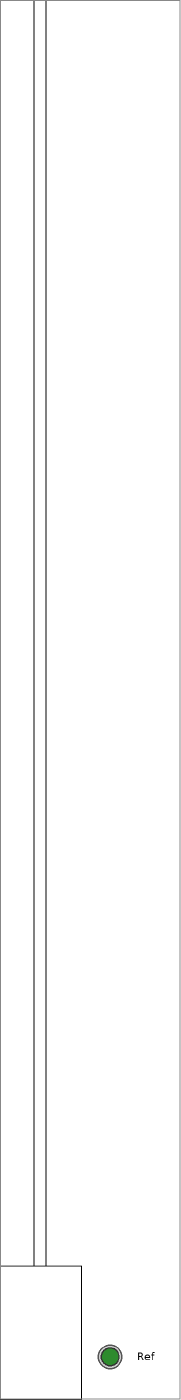
VISUALIZATION Lift_Axis  // 189x1460
VAR_IN_OUT
	Position : REAL;
	RefSensor : BOOL;
END_VAR
    Rectangle (35,0 13x1460)
    Lamp1 (100,1400 30x30), variable: RefSensor, style: Lamp-Lamp1-Green
    Rectangle (0,1320 85x140)
        p2738717112: - (1320.0 / 100.0 * Position)
    Label (140,1400 49x30), "Ref"
END_VISUALIZATION

// ---- 7_Visu/Common/Lift_Floors.TcVIS
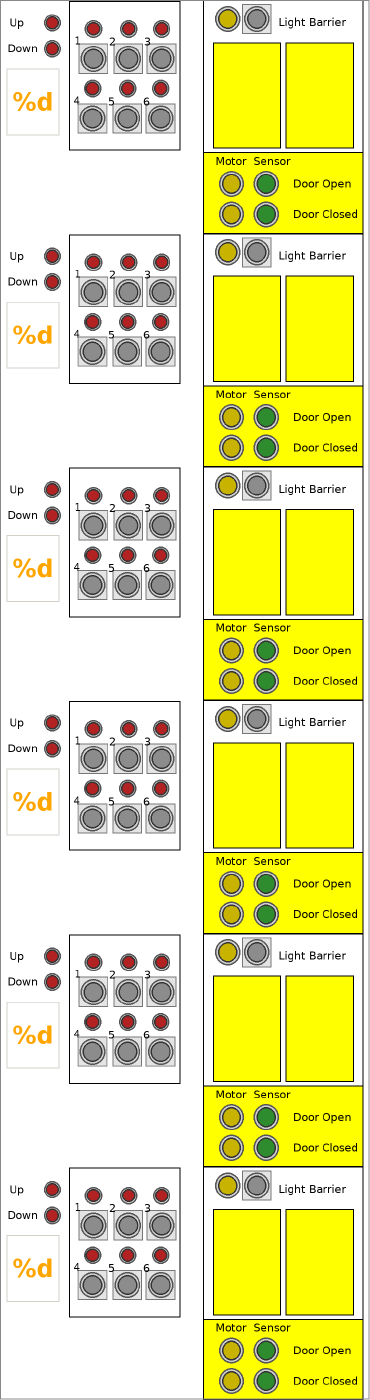
VISUALIZATION Lift_Floors  // 376x1422
VAR_IN_OUT
	Color 			: DWORD;
	Door_1_Position	: REAL;
	Door_1_M_Open	: BOOL;
	Door_1_M_Close	: BOOL;
	Door_2_Position	: REAL;
	
	Door_2_M_Open	: BOOL;
	Door_2_M_Close	: BOOL;
	Door_3_Position	: REAL;
	
	Door_3_M_Open	: BOOL;
	Door_3_M_Close	: BOOL;
	Door_4_Position	: REAL;
	
	Door_4_M_Open	: BOOL;
	Door_4_M_Close	: BOOL;
	Door_5_Position	: REAL;
	
	Door_5_M_Open	: BOOL;
	Door_5_M_Close	: BOOL;
	Door_6_Position	: REAL;
	
	Door_6_M_Open	: BOOL;
	Door_6_M_Close	: BOOL;
	
	LED_Up_1 		: BOOL;
	LED_Down_1 		: BOOL;
	FloorNumber_1 	: INT;
	BtnLed_1 		: ARRAY[1..6] OF BOOL;;
	Btn_1			: ARRAY[1..6] OF BOOL;
	LB_1 			: BOOL;
	LED_DoorOpen_1 	: BOOL;
	LED_DoorClosed_1: BOOL;

	LED_Up_2 		: BOOL;
	LED_Down_2 		: BOOL;
	FloorNumber_2 	: INT;
	BtnLed_2 		: ARRAY[1..6] OF BOOL;;
	Btn_2			: ARRAY[1..6] OF BOOL;
	LB_2 			: BOOL;
	LED_DoorOpen_2 	: BOOL;
	LED_DoorClosed_2: BOOL;


	LED_Up_3 		: BOOL;
	LED_Down_3 		: BOOL;
	FloorNumber_3 	: INT;
	BtnLed_3 		: ARRAY[1..6] OF BOOL;;
	Btn_3			: ARRAY[1..6] OF BOOL;
	LB_3 			: BOOL;
	LED_DoorOpen_3 	: BOOL;
	LED_DoorClosed_3: BOOL;

	LED_Up_4 		: BOOL;
	LED_Down_4 		: BOOL;
	FloorNumber_4 	: INT;
	BtnLed_4 		: ARRAY[1..6] OF BOOL;;
	Btn_4			: ARRAY[1..6] OF BOOL;
	LB_4 			: BOOL;
	LED_DoorOpen_4 	: BOOL;
	LED_DoorClosed_4: BOOL;

	LED_Up_5 		: BOOL;
	LED_Down_5 		: BOOL;
	FloorNumber_5 	: INT;
	BtnLed_5 		: ARRAY[1..6] OF BOOL;;
	Btn_5			: ARRAY[1..6] OF BOOL;
	LB_5 			: BOOL;
	LED_DoorOpen_5 	: BOOL;
	LED_DoorClosed_5: BOOL;

	LED_Up_6 		: BOOL;
	LED_Down_6 		: BOOL;
	FloorNumber_6 	: INT;
	BtnLed_6 		: ARRAY[1..6] OF BOOL;;
	Btn_6			: ARRAY[1..6] OF BOOL;
	LB_6 			: BOOL;
	LED_DoorOpen_6 	: BOOL;
	LED_DoorClosed_6: BOOL;

END_VAR
    Frame (0,1185 376x237)
        shows Floor(Color := Color, LED_Up := LED_Up_1, LED_Down := LED_Down_1, FloorNumber := FloorNumber_1, BtnLed := BtnLed_1, Btn := Btn_1, LB := LB_1, LED_DoorOpen := LED_DoorOpen_1, LED_DoorClosed := LED_DoorClosed_1, PositionDoor := Door_1_Position, M_Open := Door_1_M_Open, M_Close := Door_1_M_Close)
    Frame (0,948 376x237)
        shows Floor(Color := Color, LED_Up := LED_Up_2, LED_Down := LED_Down_2, FloorNumber := FloorNumber_2, BtnLed := BtnLed_2, Btn := Btn_2, LB := LB_2, LED_DoorOpen := LED_DoorOpen_2, LED_DoorClosed := LED_DoorClosed_2, PositionDoor := Door_2_Position, M_Open := Door_2_M_Open, M_Close := Door_2_M_Close)
    Frame (0,711 376x237)
        shows Floor(Color := Color, LED_Up := LED_Up_3, LED_Down := LED_Down_3, FloorNumber := FloorNumber_3, BtnLed := BtnLed_3, Btn := Btn_3, LB := LB_3, LED_DoorOpen := LED_DoorOpen_3, LED_DoorClosed := LED_DoorClosed_3, PositionDoor := Door_3_Position, M_Open := Door_3_M_Open, M_Close := Door_3_M_Close)
    Frame (0,474 376x237)
        shows Floor(Color := Color, LED_Up := LED_Up_4, LED_Down := LED_Down_4, FloorNumber := FloorNumber_4, BtnLed := BtnLed_4, Btn := Btn_4, LB := LB_4, LED_DoorOpen := LED_DoorOpen_4, LED_DoorClosed := LED_DoorClosed_4, PositionDoor := Door_4_Position, M_Open := Door_4_M_Open, M_Close := Door_4_M_Close)
    Frame (0,237 376x237)
        shows Floor(Color := Color, LED_Up := LED_Up_5, LED_Down := LED_Down_5, FloorNumber := FloorNumber_5, BtnLed := BtnLed_5, Btn := Btn_5, LB := LB_5, LED_DoorOpen := LED_DoorOpen_5, LED_DoorClosed := LED_DoorClosed_5, PositionDoor := Door_5_Position, M_Open := Door_5_M_Open, M_Close := Door_5_M_Close)
    Frame (0,0 376x237)
        shows Floor(Color := Color, LED_Up := LED_Up_6, LED_Down := LED_Down_6, FloorNumber := FloorNumber_6, BtnLed := BtnLed_6, Btn := Btn_6, LB := LB_6, LED_DoorOpen := LED_DoorOpen_6, LED_DoorClosed := LED_DoorClosed_6, PositionDoor := Door_6_Position, M_Open := Door_6_M_Open, M_Close := Door_6_M_Close)
END_VISUALIZATION

// ---- 7_Visu/Common/View_3Lifts.TcVIS
VISUALIZATION View_3Lifts  // 2x2
END_VISUALIZATION

